		rtPendantUpDownFast(CLK 	:= stCommandsIn.bPendantUpDownFast);
		ftPendantUpDownFast(CLK 	:= stCommandsIn.bPendantUpDownFast);	
		bChangeSpeedUpDown			S= (rtPendantUpDownFast.Q OR ftPendantUpDownFast.Q);
		bChangeSpeedUpDown			R= NOT CartesianZAxisRef.Status.Moving;
	
 CASE 	diManualModeCase OF
	 
		 0:
	mcCatcherHalt.Execute								:=	FALSE;	 
		 
	 	//Ruchy manualne
	mcCartesianYManualMove.JogForward					:= NOT mcCartesianYManualMove.JogBackwards AND NOT bChangeSpeedRightLeft AND
															(bManualCartesianYJogPlus OR stCommandsIn.bPendantRightwardMovement);
	mcCartesianYManualMove.JogBackwards					:= NOT mcCartesianYManualMove.JogForward AND NOT bChangeSpeedRightLeft AND
															(bManualCartesianYJogMinus OR stCommandsIn.bPendantLeftwardMovement);
	mcCartesianYManualMove.Velocity						:= SEL(stCommandsIn.bPendantRightLeftFast, 5.0, 50.0); 
                                            			
	mcCartesianZManualMove.JogForward					:= NOT mcCartesianZManualMove.JogBackwards AND NOT bChangeSpeedUpDown AND
															(bManualCartesianZJogPlus OR stCommandsIn.bPendantUpwardMovement);
	mcCartesianZManualMove.JogBackwards					:= NOT mcCartesianZManualMove.JogForward AND NOT bChangeSpeedUpDown AND
															(bManualCartesianZJogMinus OR stCommandsIn.bPendantDownwardMovement);
	mcCartesianZManualMove.Velocity						:= SEL(stCommandsIn.bPendantUpDownFast, 5.0, 50.0); 
	                                        			
	mcPreScrewerManualMove.JogForward					:= bManualPreScrewerJogPlus;
	mcPreScrewerManualMove.JogBackwards					:= bManualPreScrewerJogMinus;
	mcPreScrewerManualMove.Velocity						:= 90;
                                            			
	mcCatcherManualMove.JogForward						:= bManualCatcherJogPlus;
	mcCatcherManualMove.JogBackwards					:= bManualCatcherJogMinus;
	mcCatcherManualMove.Velocity						:= 15; 
	                                        			
	bCapSucker[1]											:= bManualCapSucker1;	
	bCapSucker[2]											:= bmanualCapSucker2;	
	bCapSucker[3]											:= bManualCapSucker3;	
	bCapSucker[4]											:= bManualCapSucker4;	
	                          	    					                     
	bCapBlower1											:= bManualCapBlower1;	
	bCapBlower2											:= bManualCapBlower2;	
	bCapBlower3											:= bManualCapBlower3;	
	bCapBlower4											:= bManualCapBlower4;	
	                          		    				                 
	bCapCatcher1										:= bManualCapCatcher1;
	bCapCatcher2										:= bManualCapCatcher2;
	bCapCatcher3										:= bManualCapCatcher3;
	bCapCatcher4					    				:= bManualCapCatcher4;
	
	
	
	IF bManualStrawCatchersOpen	THEN
		bStrawCatchersOpen								:= TRUE;
		bStrawCatchersClose								:= FALSE;
		bManualStrawCatchersClose						:= FALSE;
	END_IF	                                    		
                                                		
	IF bManualStrawCatchersClose	THEN        		
		bStrawCatchersOpen								:= FALSE;
		bStrawCatchersClose								:= TRUE;
		bManualStrawCatchersOpen						:= FALSE;
	END_IF		                                		
	                                            		
     IF bManualStrawCatcherActuatorOut THEN     		
		 bStrawCatcherActuatorOut						:= TRUE;
		 bStrawCatcherActuatorIn						:= FALSE;
		 bManualStrawCatcherActuatorIn					:= FALSE;
	 END_IF                                     		
	                                            	
     IF bManualStrawCatcherActuatorIn THEN      	
		 bStrawCatcherActuatorIn						:= TRUE;
		 bStrawCatcherActuatorOut						:= FALSE;
		 bManualStrawCatcherActuatorOut					:= FALSE;
	 END_IF
	 
	 //Zaczynam sekwencje 
	 IF trStepButton.Q THEN
		 VirtualEna											:= TRUE;
		 ResetCommands();
		 bCapCatcher1										:= FALSE;
		 bCapCatcher2										:= false;
		 bCapCatcher3										:= false;
		 bCapCatcher4										:= false;
		 bCartesianReady									:= bCartesianInHomePos;
		 diManualModeCase									:= diManualModeCase + 10;
	 END_IF
	 
	 IF rtSetEncoderOffsetAxisZ.Q THEN
		diManualModeCase									:= diManualModeCase + 500;
	 END_IF
 
 
 		10:	//Dojazd do poz home
	bStepButton												:= TRUE;
	                                                    	
	mcCartesianZMoveAbsolute.Execute						:= NOT bAxisZInHomePos;		
	mcCartesianZMoveAbsolute.Position						:= 420;
	mcCartesianZMoveAbsolute.Acceleration					:= 200.0;
	mcCartesianZMoveAbsolute.Deceleration					:= 200.0;
	mcCartesianZMoveAbsolute.Velocity						:= 30;
	                                        				
	//najpierw os Z potem winda chwytakow   				
	mcCatcherMoveAbsolute.Execute							:= NOT bAxisStrawCatcherHomePos AND bAxisZInHomePos;		
	mcCatcherMoveAbsolute.Position							:= stParameters.lrCatcherCatchingPosition;
	mcCatcherMoveAbsolute.Acceleration						:= 200.0;
	mcCatcherMoveAbsolute.Deceleration						:= 200.0;
	mcCatcherMoveAbsolute.Velocity							:= 30;
	                                        				
	mcCartesianYMoveAbsolute.Execute						:= NOT bAxisYInHomePos AND bAxisZInHomePos;
	mcCartesianYMoveAbsolute.Position						:= stParameters.lrPickYPosition;
	mcCartesianYMoveAbsolute.Acceleration					:= 200.0;
	mcCartesianYMoveAbsolute.Deceleration					:= 200.0;
	mcCartesianYMoveAbsolute.Velocity						:= 30; 
	                                                    	
	IF bAxisZInHomePos THEN
		GVL_VIS.bCapSorterPreScrewerCatchStationHoming			:= NOT fbStrawCatcherLift.bHomingDone;
		GVL_VIS.bCapSorterPreScrewerCatcherStationHeightSet		:= NOT GVL_VIS.bCapSorterPreScrewerCatchStationHoming AND NOT bStrawCatcherLiftInHomePos;
		bEnableLift												:= GVL_VIS.bCapSorterPreScrewerCatcherStationHeightSet;
	END_IF

		IF 	bCartesianInHomePos AND bStrawCatcherLiftInHomePos THEN
			mcCartesianZMoveAbsolute.Execute              	:= FALSE;
			mcCatcherMoveAbsolute.Execute                 	:= FALSE;
			mcCartesianYMoveAbsolute.Execute              	:= FALSE;
			GVL_VIS.bCapSorterPreScrewerCatchStationHoming	:= FALSE;
			diManualModeCase								:= diManualModeCase + 5;
		END_IF
		
		15: //Ustaw obracarkę w pozycji
	bStepButton												:= TRUE;
	                                                    	
	mcPreScrewerMoveRelative.Execute						:= TRUE;
	mcPreScrewerMoveRelative.Distance						:=  -1 * DINT_TO_LREAL(LREAL_TO_DINT(PreScrewerAxisRef.NcToPlc.SetPos) MOD 360);
	mcPreScrewerMoveRelative.Acceleration					:= 200.0;
	mcPreScrewerMoveRelative.Deceleration					:= 200.0;
	mcPreScrewerMoveRelative.Velocity						:= 180.0;	
	                                                    	
		IF mcPreScrewerMoveRelative.Done THEN           	
			mcPreScrewerMoveRelative.Execute				:= FALSE;
			
			IF bCartesianReady THEN
				diManualModeCase							:= diManualModeCase + 10;
			ELSE	                                        
				bStepButton									:= FALSE;
				diManualModeCase							:= diManualModeCase + 5;
			END_IF
			
		END_IF	

		
//--------------------------------jazda na poz pick------------------------------------------------------------------			
		20:	//Kolejny krok
	 IF trStepButton.Q THEN
		diManualModeCase									:= diManualModeCase + 5;
	 END_IF

		25:
	bStepButton												:= TRUE;
	
	mcCartesianZMoveAbsolute.Execute						:= TRUE;		
	mcCartesianZMoveAbsolute.Position						:= stParameters.lrPickZPosition;
	
		IF mcCartesianZMoveAbsolute.Done THEN
			mcCartesianZMoveAbsolute.Execute				:= FALSE;
			bStepButton										:= FALSE;
			diManualModeCase								:= diManualModeCase + 5;
		END_IF

		
//----------------------------Sekwencyjne zalączanie ssawek----------------------------------------------------------------	
		30: //Kolejny krok
	 IF trStepButton.Q THEN
		FOR i:=1 TO 4 DO
			bCapSucker[i]									:= TRUE;
		END_FOR	 
	 
		diManualModeCase									:= diManualModeCase + 5;
	 END_IF
		
		35: //Załączanie ssawek
	tonVacuumWatchdog.IN									:= TRUE;
	bStepButton												:= TRUE;

	
	
		IF tonVacuumWatchdog.Q THEN	
			bStepButton										:= FALSE;		 
			tonVacuumWatchdog.IN							:= FALSE;								
			diManualModeCase								:= diManualModeCase + 20;				
		END_IF
		
		
//-------------------------------Dojazd do pozycji zamykania wings'ów-------------------------------------------------------------------			
		55: //Kolejny krok
	 IF trStepButton.Q THEN
		diManualModeCase									:= diManualModeCase + 5;
	 END_IF	
	 
	 	60:
	bStepButton												:= TRUE;	
	mcCartesianZMoveAbsolute.Execute						:= TRUE;		
	mcCartesianZMoveAbsolute.Position						:= stParameters.lrCapCatcherZPosition;	
		
		IF mcCartesianZMoveAbsolute.Done THEN
			
			FOR i:=1 TO 4 DO
				bCapSucker[i]								R= NOT  bCapSucker[i];
			END_FOR 
			
			bStepButton										:= FALSE;	
			mcCartesianZMoveAbsolute.Execute				:= FALSE;
			diManualModeCase								:= diManualModeCase + 5;		
		END_IF

		
//--------------------------------Zamykanie vings'ów------------------------------------------------------------------			
		65://Kolejny krok
	 IF trStepButton.Q THEN
		diManualModeCase									:= diManualModeCase + 5;
	 END_IF	
	 
	 	70:
	bStepButton												:= FALSE;	
	bCapCatcher1											:= TRUE;
	bCapCatcher2											:= TRUE;
	bCapCatcher3											:= TRUE;
	bCapCatcher4											:= TRUE;
	diManualModeCase										:= diManualModeCase + 5;

	
//---------------------------------dojazd do poz. Top-----------------------------------------------------------------			
		75://Kolejny krok
	 IF trStepButton.Q THEN
		diManualModeCase									:= diManualModeCase + 5;
	 END_IF	
		
		80:
	bStepButton												:= TRUE;
	mcCartesianZMoveAbsolute.Execute						:= TRUE;
	mcCartesianZMoveAbsolute.Position						:= stParameters.lrTopZPosition;
		
		IF mcCartesianZMoveAbsolute.Done THEN
			bStepButton										:= FALSE;	
			mcCartesianZMoveAbsolute.Execute				:= FALSE;
			diManualModeCase								:= diManualModeCase + 5;		
		END_IF

		
//-----------------------------------dojazd osi Y do pozycji place---------------------------------------------------------------			
		85://Kolejny krok
	 IF trStepButton.Q THEN
		diManualModeCase									:= diManualModeCase + 5;
	 END_IF	
	 
	 90:
	bStepButton												:= TRUE;
	mcCartesianYMoveAbsolute.Execute						:= TRUE;
	mcCartesianYMoveAbsolute.Position						:= stParameters.lrPlaceYPosition;
	
	 mcCartesianZMoveAbsolute.Execute						:= CartesianYAxisRef.NcToPlc.ActPos > stParameters.lrPickYPosition + 50.0;
	 mcCartesianZMoveAbsolute.Position						:= stParameters.lrCartesianCatchZPosition;
	 
		IF mcCartesianYMoveAbsolute.Done AND mcCartesianZMoveAbsolute.Done THEN
			bStepButton										:= FALSE;
			mcCartesianYMoveAbsolute.Execute				:= FALSE;
			GVL_VIS.bCapSorterPreScrewerBottleCatcherCatch	:= TRUE;					//Zamykanie chwytaków butelek
			diManualModeCase								:= diManualModeCase + 10;
		END_IF		
		
		
		
		

		
//-------------------------------Wybór pracy: słomka albo fliptop & sterowanie krabami------------------------	
		100://Kolejny krok
	 IF trStepButton.Q THEN
		diManualModeCase									:= diManualModeCase + 5;
	 END_IF	
	 
		105://Ustaw pozycję wirtualnej osi tak samo jak na osi Z
	fbVirtualAxis.fPosition									:= CartesianZAxisRef.NcToPlc.ActPos;
	fbVirtualAxis.SetPosAbsClearLag(bExecute				:= TRUE);
		
		IF fbVirtualAxis.pSetPos.Busy THEN
			diManualModeCase								:= diManualModeCase + 1;
		ELSIF fbVirtualAxis.pSetPos.Error OR fbVirtualAxis.pSetPos.CommandAborted THEN
    		udiErrorID										:= 6;
    		udiErrorID										:= udiErrorID + iStationIndex;
    		sErrorDescription								:= 'Błąd podnosnika lub brak zasilania';
    		sErrorDescription2								:= ' ';	
		END_IF
		
		106:
	fbVirtualAxis.SetPosAbsClearLag(bExecute				:= FALSE);
		
		IF fbVirtualAxis.pSetPos.Done THEN
			diManualModeCase								:= diManualModeCase + 4;
		END_IF


		110: 	//Przy aktywowanych slomkach--> wysuń kraby
	IF stParameters.bStrawCatcherON THEN
		bStrawCatcherActuatorIn								:= FALSE;
		bStrawCatcherActuatorOut							:= TRUE; 
		diManualModeCase									:= diManualModeCase + 1;
	ELSE
			//przeskakuję do sprawdzania czy mam szukanie gwintu
		bStrawCatcherActuatorIn								:= TRUE;
		bStrawCatcherActuatorOut							:= FALSE; 			
		fbGearInAxisZ.Enable								:= TRUE;
		
			IF fbGearInAxisZ.InGear THEN
				fbGearInAxisZ.Enable						:= FALSE;
				IF stParameters.lrScrewFinding > 0 THEN
			 		diManualModeCase						:= diManualModeCase + 26;
		 		ELSE
					diManualModeCase						:= diManualModeCase + 30;
			 	END_IF
			 END_IF
	END_IF
		
		
		111://zamknij kraby
	bStepButton												:= TRUE;	
	bStrawCatchersOpen										:= NOT bStrawCatcherOut;
	bStrawCatchersClose										:= bStrawCatcherOut;
	
		//zamkniete kraby
		IF tonStrawCatcher1Close.Q (*AND tonStrawCatcher2Close.Q*) AND tonStrawCatcher3Close.Q AND tonStrawCatcher4Close.Q THEN
			bStepButton										:= FALSE;
			diManualModeCase								:= diManualModeCase + 4;
		END_IF

		
//-----------------------------------Prowadzenie slomki do pozycji wspolnego ruchu-------------------------------			
		115://Kolejny krok
	 IF trStepButton.Q THEN
		diManualModeCase									:= diManualModeCase + 5;
	 END_IF			
		
		120://gear'owanie napędu prowadzenia słomki
	fbGearInCatcherAxis.Enable								:= TRUE;
	fbGearInCatcherAxis.GearRatio							:= 1;
	fbGearInAxisZ.Enable									:= TRUE;
	fbGearInAxisZ.GearRatio									:= 0.0000000001;
	bStepButton												:= TRUE;
		
		IF fbGearInCatcherAxis.InGear AND fbGearInAxisZ.InGear THEN
			//fbGearInCatcherAxis.Enable						:= FALSE;
			//fbGearInAxisZ.Enable							:= FALSE;
			diManualModeCase								:= diManualModeCase + 10;
		END_IF

		
//-----------------------------------Prowadzenie, wkładanie nasadki oraz rozgirowanie osi do prowadzenia słomki------------------------------------------			
		130: 
	fbVirtualAxis.fPosition									:= (stParameters.LrCheckStrawCatcherActuatorZPosition - stParameters.lrStrawInsertDistance);	//Pozycja sprawdzania cofnięcia krabów
	fbVirtualAxis.fVelocity									:= 100.0;	//10
	fbVirtualAxis.fAcceleration								:= 1000.0;
	fbVirtualAxis.fDeceleration								:= 1000.0;
	fbVirtualAxis.fJerk										:= 10000.0;			
			
	bStepButton												:= TRUE;
	bVirtualMove											:= TRUE;				
//	fbGearInAxisZ.Execute									:= CatcherAxisRef.NcToPlc.ActPos <= (stParameters.lrCatcherPlacePosition + stParameters.lrStrawInsertDistance);

	//IF CatcherAxisRef.NcToPlc.ActPos <= (stParameters.lrCatcherCatchingPosition - stParameters.lrStrawInsertDistance) THEN
	//	fbGearInAxisZ.GearRatio								:= 1;
	//END_IF
	
	IF (CatcherAxisRef.NcToPlc.ActPos + stParameters.lrCatcherHightSV) <= (stParameters.lrCartesianCatchZPosition-(stParameters.lrCapHight + 25)) THEN
		fbGearInAxisZ.GearRatio								:= 1;
	END_IF
	
			//Otwórz chwytaki słomek
		IF CartesianZAxisRef.NcToPlc.ActPos <= stParameters.lrStrawCatcherZPosition THEN					
			bStrawCatchersOpen								:= TRUE;
			bStrawCatchersClose								:= FALSE;
		END_IF
		
		// 10mm stały offset - wysokość nad butelką
		IF (CatcherAxisRef.NcToPlc.ActPos <= 1.0) OR (CatcherAxisRef.NcToPlc.ActPos + 32 <= ((stParameters.lrBottleHight + 10.0) - stParameters.lrCatcherHightSV)) THEN	//13 20
			fbGearInCatcherAxis.GearRatio					:= 0.0000000001;
		END_IF
	
			IF tonStrawCatcher1Open.Q AND tonStrawCatcher2Open.Q AND tonStrawCatcher3Open.Q AND tonStrawCatcher4Open.Q THEN																				
				//Cofnij chwytaki słomek
				bStrawCatcherActuatorIn						:= TRUE;
				bStrawCatcherActuatorOut					:= FALSE;				
			END_IF			
			
				IF stVirtualMove_Out.Done THEN
					//fbGearInAxisZ.Enable					:= FALSE;
					//fbGearOutCatcherAxis.Execute			:= FALSE;
					fbGearInCatcherAxis.GearRatio				:= 0.0000000001;
					bVirtualMove							:= FALSE;	
					bStepButton								:= FALSE;
					diManualModeCase						:= diManualModeCase + 5;
				END_IF					
		
//------------------------------------Zakończenie wkładania nasadki---------------------------------------------------			
		135://Kolejny krok
		//mcCatcherHalt.Execute								:=	FALSE;
		
	 IF trStepButton.Q THEN
		 IF stParameters.lrScrewFinding > 0 THEN
			 diManualModeCase								:= diManualModeCase + 1;
		 ELSE
			 diManualModeCase								:= diManualModeCase + 5;
		 END_IF
		
	 END_IF	

//------------------------------------Szukanie gwintu---------------------------------------------------				 	
		136:
	fbVirtualAxis.fVelocity									:= 800.0;	//10
	fbVirtualAxis.fAcceleration								:= 1000.0;
	fbVirtualAxis.fDeceleration								:= 1000.0;
	fbVirtualAxis.fJerk										:= 10000.0;			
		
	fbVirtualAxis.fPosition									:= stParameters.lrScrewerStartZPosition;
	bVirtualMove											:= TRUE;
	bStepButton												:= TRUE;	
	
		IF stVirtualMove_Out.Done THEN
			bCapSucker[1]										:= FALSE;
			bCapSucker[2]										:= FALSE;
			bCapSucker[3]										:= FALSE;
			bCapSucker[4]										:= FALSE;

			mcPreScrewerMoveRelative.Distance				:= stParameters.lrScrewFinding * -1.0;
			mcPreScrewerMoveRelative.Acceleration			:= stParameters.lrScrewAcceleration;
			mcPreScrewerMoveRelative.Deceleration			:= stParameters.lrScrewAcceleration;
			mcPreScrewerMoveRelative.Velocity				:= stParameters.lrScrewSpeed;
			mcPreScrewerMoveRelative.Execute				:= TRUE;
		END_IF
		
				IF mcPreScrewerMoveRelative.Done OR ABS(PreScrewerAxisRef.NcToPlc.PosDiff) > 60.0 OR mcPreScrewerMoveRelative.Error THEN
					bVirtualMove							:= FALSE;
					bStepButton								:= FALSE;
					mcPreScrewerMoveRelative.Execute		:= FALSE;
					diManualModeCase						:= diManualModeCase + 1;
				END_IF	
		
		137://Kolejny krok
	 IF trStepButton.Q THEN
		 diManualModeCase									:= diManualModeCase + 3;		
	 END_IF					
	 
	 	140:
	lrPreScrewerAxisSavedPosition							:= PreScrewerAxisRef.NcToPlc.ActPos;	//zapisywanie pozycji przed zakrecaniem		
	fbVirtualAxis.fPosition									:= stParameters.lrPlaceZPosition - stParameters.lrStrawInsertDistance;
	fbVirtualAxis.fVelocity									:= stParameters.lrCatcherSpeed;
	fbVirtualAxis.fAcceleration								:= 1000.0;
	fbVirtualAxis.fDeceleration								:= 1000.0;
	fbVirtualAxis.fJerk										:= 10000.0;
	bVirtualMove											:= TRUE;
	bStepButton												:= TRUE;
	
		IF CartesianZAxisRef.NcToPlc.ActPos <= stParameters.lrScrewerStartZPosition + 1.0 THEN
			bCapSucker[1]										:= FALSE;
			bCapSucker[2]										:= FALSE;
			bCapSucker[3]										:= FALSE;
			bCapSucker[4]										:= FALSE;
			mcPreScrewerMoveRelative.Execute				:= TRUE;
			mcPreScrewerMoveRelative.Distance				:= stParameters.lrScrewDistance;
			mcPreScrewerMoveRelative.Acceleration			:= stParameters.lrScrewAcceleration;
			mcPreScrewerMoveRelative.Deceleration			:= stParameters.lrScrewAcceleration;
			mcPreScrewerMoveRelative.Velocity				:= stParameters.lrScrewSpeed;// do bylo 600.0;//stParameters.lrScrewSpeed;
			diManualModeCase								:= diManualModeCase + 5;			
		END_IF

	
		145:
	bStepButton												:= TRUE;
	
			//otwórz centrowniki butelek
		IF (GVL_Recipe.bCapSorterPreScrewerCatchAngleOpenEnaShow AND
			ABS(PreScrewerAxisRef.NcToPlc.ActPos - lrPreScrewerAxisSavedPosition) >= GVL_Recipe.lrCapSorterPreScrewerCatchAngleOpenSV) THEN
			bBottleCatcherCatchTemp					:= FALSE;
		END_IF
	
		IF PreScrewerAxisRef.NcToPlc.PosDiff > 100.0 OR (stVirtualMove_Out.Done AND mcPreScrewerMoveRelative.Done) THEN
			bBottleCatcherCatchTemp							:= FALSE;
			bCapCatcher1									:= FALSE;
		 	bCapCatcher2									:= FALSE;
		 	bCapCatcher3									:= FALSE;
		 	bCapCatcher4									:= FALSE;
			bVirtualMove									:= FALSE;
			bCapsBlowON										:= TRUE;
			
				IF fbVirtualAxis.bMoving THEN
					fbVirtualAxis.Halt(bExecute := TRUE);
				ELSE
					fbVirtualAxis.Halt(bExecute := FALSE);
					diManualModeCase						:= diManualModeCase + 5;
				END_IF	
				
		END_IF
		
		150:
	bStepButton												:= TRUE;	
	fbVirtualAxis.fPosition									:= stParameters.lrPlaceZPosition + 20.0;	
	fbVirtualAxis.fVelocity									:= 800.0;//10.0;
	fbVirtualAxis.fAcceleration								:= 1000.0;
	fbVirtualAxis.fDeceleration								:= 1000.0;
	fbVirtualAxis.fJerk										:= 10000.0;
	bVirtualMove											:= TRUE;
	fbGearInCatcherAxis.Enable								:= FALSE;
	fbGearInAxisZ.Enable									:= FALSE;
	
		IF stVirtualMove_Out.Done THEN
			bVirtualMove									:= FALSE;
			diManualModeCase								:= diManualModeCase + 5;
		END_IF
		
		
					151:		//na testy do usunięcia
					fbVirtualAxis.fPosition									:= CartesianZAxisRef.NcToPlc.ActPos;
					fbVirtualAxis.SetPosAbsClearLag(bExecute				:= TRUE);
					
					152:
					fbVirtualAxis.SetPosAbsClearLag(bExecute				:= FALSE);
	
	
		155:
	fbGearOutAxisZ.Execute									:= TRUE;
	fbGearOutCatcherAxis.Execute							:= TRUE;
	
		IF NOT CartesianZAxisRef.Status.Coupled AND NOT CatcherAxisRef.Status.Coupled THEN
			fbGearOutAxisZ.Execute							:= FALSE;
			fbGearOutCatcherAxis.Execute					:= FALSE;
			bStepButton										:= FALSE;
			diManualModeCase								:= diManualModeCase + 5;
		END_IF

//-------------------------------------Dojazd do poz home---------------------------------------------			
		160://Kolejny krok
	 IF trStepButton.Q THEN
		diManualModeCase									:= diManualModeCase + 5;
	 END_IF	
		
		165:
	GVL_VIS.bCapSorterPreScrewerBottleCatcherCatch	:= FALSE;	
	bStepButton										:= TRUE;	
	mcCartesianZMoveAbsolute.Execute				:= TRUE;		
	mcCartesianZMoveAbsolute.Position				:= stParameters.lrTopZPosition;
                                            		
	mcCartesianYMoveAbsolute.Execute				:= ABS(mcCartesianZMoveAbsolute.Position - stParameters.lrTopZPosition) <= 1.0;
	mcCartesianYMoveAbsolute.Position				:= stParameters.lrPickYPosition;
	                                        		
	mcPreScrewerMoveRelative.Execute				:= mcCartesianYMoveAbsolute.Done;
	mcPreScrewerMoveRelative.Velocity				:= 180.0;
	mcPreScrewerMoveRelative.Distance				:= -1 * DINT_TO_LREAL(LREAL_TO_DINT(PreScrewerAxisRef.NcToPlc.SetPos) MOD 360);
	                                        		
	mcCatcherMoveAbsolute.Execute					:= mcCartesianZMoveAbsolute.Done;		
	mcCatcherMoveAbsolute.Position					:= stParameters.lrCatcherCatchingPosition;
	
		IF (mcCartesianZMoveAbsolute.Done AND mcCartesianYMoveAbsolute.Done
			AND mcPreScrewerMoveRelative.Done AND mcCatcherMoveAbsolute.Done) THEN
				bCapsBlowON							:= TRUE;
				bStepButton							:= FALSE;
				ResetCommands();            		
				diManualModeCase					:= 0;
		END_IF	 
		
		
	500: //Ustawianie offsetu na soi Z kartezjana
	bCartesianZServoPower				:= FALSE;
	
	fbAxisZPositioningOffset.Position	:= 0.0;
	fbAxisZPositioningOffset.Execute	:= NOT CartesianZAxisRef.Status.Disabled;
	
	IF fbAxisZPositioningOffset.Busy THEN
		diManualModeCase				:= diManualModeCase + 5;
	END_IF
		
	505:
	IF NOT fbAxisZPositioningOffset.Busy THEN
		fbAxisZPositioningOffset.Execute := FALSE;
		bCartesianZServoPower			 := TRUE;
		diManualModeCase				:= diManualModeCase + 5;
	END_IF
	
	510:
	IF 	mcCartesianZPower.Status THEN
		diManualModeCase				:= 0;
	END_IF
		
 END_CASE
END_ACTION

ACTION PreparingToDisable:
//BAZOWANIE 

mcCartesianYPower.Override				:=	100;			
mcCartesianZPower.Override				:=	100;			
mcPreScrewerPower.Override				:=	100;			
mcCatcherPower.Override					:=	100;	

bCartesianYServoPower					:= TRUE;
bCartesianZServoPower					:= TRUE;
bPreScrewerPower						:= TRUE;
bCatcherPower							:= TRUE;	

mcCartesianYManualMove.JogBackwards		:=FALSE;
mcCartesianZManualMove.JogBackwards		:=FALSE;
mcPreScrewerManualMove.JogBackwards		:=FALSE;
mcCatcherManualMove.JogBackwards		:=FALSE;

mcCartesianYManualMove.JogForward		:=FALSE;
mcCartesianZManualMove.JogForward		:=FALSE;
mcPreScrewerManualMove.JogForward		:=FALSE;
mcCatcherManualMove.JogForward			:=FALSE;
bCycleNotDone							:= FALSE;



IF mcCartesianYPower.Status AND mcCartesianZPower.Status AND mcPreScrewerPower.Status AND mcCatcherPower.Status THEN
		
		CASE iDisablingCase OF
		
			0:
				iDisablingCase							:= iDisablingCase	+	10;
			
			10: 

				//Otwórz chwytaki
				bCapCatcher1				:= FALSE;
				bCapCatcher2				:= FALSE;
				bCapCatcher3				:= FALSE;
				bCapCatcher4				:= FALSE;
				//Wyłącz ssawki
				bCapSucker[1]				:= FALSE;
				bCapSucker[2]				:= FALSE;
				bCapSucker[3]				:= FALSE;
				bCapSucker[4]				:= FALSE;
				//Wyłącz odmuchy
				bCapBlower1					:= FALSE;
				bCapBlower2					:= FALSE;
				bCapBlower3					:= FALSE;
				bCapBlower4					:= FALSE;
				//Otwórz chwytaki słomek
				bStrawCatchersOpen			:= TRUE;
				bStrawCatchersClose			:= FALSE;
				//Cofnij chwytaki słomek
				bStrawCatcherActuatorIn		:= TRUE;
				bStrawCatcherActuatorOut	:= FALSE;
				//Podjedź robotem i chwytakiem słomek w górę jak cofnięty chwytak słomek - bazuj podnośnik Jisang
				IF tonStrawCatcherIn.Q THEN	
					mcCartesianZMoveAbsolute.Execute		:= TRUE;		
					mcCartesianZMoveAbsolute.Position		:= 420;//stParameters.lrTopZPosition;
					mcCartesianZMoveAbsolute.Acceleration	:= stParameters.lrPickerAcceleration;
					mcCartesianZMoveAbsolute.Deceleration	:= stParameters.lrPickerAcceleration;
					mcCartesianZMoveAbsolute.Velocity		:= 30;//stParameters.lrPickerSpeed;
					
					mcCatcherMoveAbsolute.Execute			:= TRUE;		
					mcCatcherMoveAbsolute.Position			:= stParameters.lrCatcherCatchingPosition;
					mcCatcherMoveAbsolute.Acceleration		:= stParameters.lrCatcherAcceleration;
					mcCatcherMoveAbsolute.Deceleration		:= stParameters.lrCatcherAcceleration;
					mcCatcherMoveAbsolute.Velocity			:= 30;//stParameters.lrCatcherSpeed;

					//Następny krok
					iDisablingCase								:= iDisablingCase + 10;
				END_IF
				//Reset komendy ruchu osi X
				mcCartesianYMoveAbsolute.Execute		:= FALSE;
				
		
			20:		
	(*Czekam na pozycję Z w górze i ruszam osią poziomą X na pozycję pobierania i czekam na obie pozycje*)
				//bStrawCatcherLiftEnable						R= ABS(CartesianYAxisRef.NcToPlc.ActPos - stParameters.lrPickYPosition)<=10.0;
				
				IF (CartesianZAxisRef.NcToPlc.ActPos > stParameters.lrTopZPosition - stParameters.lrBendingDistance) OR
					mcCartesianZMoveAbsolute.Done THEN					
					//Jedź osią poziomą X na pozycję pick
					mcCartesianYMoveAbsolute.Execute		:= TRUE;
					mcCartesianYMoveAbsolute.Position		:= stParameters.lrPickYPosition;
					mcCartesianYMoveAbsolute.Acceleration	:= stParameters.lrPickerAcceleration;
					mcCartesianYMoveAbsolute.Deceleration	:= stParameters.lrPickerAcceleration;
					mcCartesianYMoveAbsolute.Velocity		:= 30;//stParameters.lrPickerSpeed;
					//Ustaw obracarkę w pozycji
					mcPreScrewerMoveRelative.Execute		:= TRUE;
					mcPreScrewerMoveRelative.Distance		:=  -1 * DINT_TO_LREAL(LREAL_TO_DINT(PreScrewerAxisRef.NcToPlc.SetPos) MOD 360);
					mcPreScrewerMoveRelative.Acceleration	:= stParameters.lrScrewAcceleration;
					mcPreScrewerMoveRelative.Deceleration	:= stParameters.lrScrewAcceleration;
					mcPreScrewerMoveRelative.Velocity		:= 180;//stParameters.lrScrewSpeed;
				END_IF
				IF mcPreScrewerMoveRelative.Done THEN
					mcPreScrewerMoveRelative.Execute		:= FALSE;
					mcPreScrewerHome(Axis := PreScrewerAxisRef, HomingMode := MC_Direct, Position := 0, Execute := TRUE);					
				END_IF
				//Jak obie pozycje osiągnięte to następny krok
				IF mcCartesianYMoveAbsolute.Done AND mcCartesianZMoveAbsolute.Done AND mcPreScrewerHome.Done AND fbStrawCatcherLift.eState =  E_Station.eDisabled THEN
					//Reset komendy ruchu osi
					mcCartesianYMoveAbsolute.Execute		:= FALSE;
					mcCartesianZMoveAbsolute.Execute		:= FALSE;
					mcPreScrewerHome.Execute				:= FALSE;
					//Wysuń chwytaki słomek jesli to potrzebuje recepta
					bStrawCatcherActuatorIn					:= TRUE;
					bStrawCatcherActuatorOut				:= FALSE;
					//Następny krok
					iDisablingCase								:= iDisablingCase + 10;
				END_IF
			
			30:	//Koniec
				eState								:= E_Station.eDisabled;
				bHomingDone							:= FALSE;
				iDisablingCase						:= 0;
		END_CASE
END_IF
END_ACTION

ACTION Reject:

CASE iRejectCase OF
	0:

		mcCartesianZMoveAbsolute.Position	:= stParameters.lrPickZPosition - lrAxisZ_RejectOffset;	
		mcCartesianZMoveAbsolute.Execute	:= NOT bTubeReject;
	
				//Przyssanie wszystkich nasadek (przypadek wcisnietej), lub pojedynczej (wykryto brak słomki)
			FOR i:=1 TO 4 DO	
				bCapSucker[i]					:=SEL(bTubeReject, stParameters.bPickerActiv[i] AND NOT tonSuckedOk[i].Q, NOT stMoverStatus.stSlotStatus[i].bTubePresent AND stParameters.bPickerActiv[i]);//SEL(bTubeReject, TRUE, NOT stMoverStatus.stSlotStatus[i].bTubePresent AND stParameters.bPickerActiv[i]);
			END_FOR
		
		iRejectCase	:= 5;
	
	
	5:
			IF bTubeReject OR mcCartesianZMoveAbsolute.Done THEN
				mcCartesianZMoveAbsolute.Execute	:= FALSE;
				iRejectCase	:= 10;
			END_IF
	
	10:
		tonVacuumWatchdog.IN					:= TRUE;
	

		
			IF bAllSlotsVacuumStatus OR tonVacuumWatchdog.Q THEN
					//Podjazd do góry
				mcCartesianZMoveAbsolute.Position	:= stParameters.lrTopZPosition;
				mcCartesianZMoveAbsolute.Execute	:= TRUE;	
				tonVacuumWatchdog.IN				:= FALSE;
				iRejectCase	:= 20;
			END_IF
	
	20:
			//Zamykanie łapek
			IF CartesianZAxisRef.NcToPlc.ActPos > stParameters.lrCapCatcherZPosition THEN
				bCapCatcher1					:= TRUE;
				bCapCatcher2					:= TRUE;
				bCapCatcher3					:= TRUE;
				bCapCatcher4					:= TRUE;
			ELSIF rtAxisZMoving.Q THEN	//oddmuch nie przyssanych nakrętek
				bCapBlow1						:= NOT bCapSucker[1];
            	bCapBlow2						:= NOT bCapSucker[2];
            	bCapBlow3						:= NOT bCapSucker[3];
            	bCapBlow4						:= NOT bCapSucker[4];
				bCapsBlowON						:= TRUE;
			END_IF
			
			IF ABS(CartesianZAxisRef.NcToPlc.ActPos - mcCartesianZMoveAbsolute.Position) <= stParameters.lrBendingDistance THEN
				mcCartesianZMoveAbsolute.Execute	:= FALSE;	
				bMissingCaps						:= TRUE;
				mcCartesianYMoveAbsolute.Position	:= 3.0;
				mcCartesianYMoveAbsolute.Execute	:= TRUE;
				
					FOR i:= 1 TO 4 DO
						bCapSucker[i]				:= FALSE;
					END_FOR				
				
				iRejectCase							:= 30;
			END_IF
		
		30:
			IF ABS(CartesianYAxisRef.NcToPlc.ActPos - mcCartesianYMoveAbsolute.Position) <= stParameters.lrBendingDistance THEN
				mcCartesianYMoveAbsolute.Execute	:= FALSE;
					IF NOT mcCartesianZMoveAbsolute.Busy THEN
						mcCartesianZMoveAbsolute.Position	:= 380.0;
						mcCartesianZMoveAbsolute.Execute	:= TRUE;	
						iRejectCase		:= 40;
					END_IF
			ELSIF ABS(CartesianYAxisRef.NcToPlc.ActPos - mcCartesianYMoveAbsolute.Position) <= 50.0 THEN	
					bCapCatcher1					:=FALSE;
					bCapCatcher2					:=FALSE;
					bCapCatcher3					:=FALSE;
					bCapCatcher4					:=FALSE;
			END_IF
			
		40:
			IF ABS(CartesianZAxisRef.NcToPlc.ActPos - mcCartesianZMoveAbsolute.Position) <= stParameters.lrBendingDistance AND NOT bCapsBlowON THEN
				bCapsBlowON						:= TRUE;
				bCapBlow1						:= TRUE;
            	bCapBlow2						:= TRUE;
            	bCapBlow3						:= TRUE;
            	bCapBlow4						:= TRUE;
				mcCartesianZMoveAbsolute.Execute	:= FALSE;	
				iRejectCase		:= 50;
			END_IF
	
		50:
			mcCartesianZMoveAbsolute2.Position		:= stParameters.lrTopZPosition;
			mcCartesianZMoveAbsolute2.Acceleration	:= stParameters.lrPickerAcceleration;
			mcCartesianZMoveAbsolute2.Deceleration	:= stParameters.lrPickerAcceleration;
			mcCartesianZMoveAbsolute2.Velocity		:= stParameters.lrPickerSpeed;
			mcCartesianZMoveAbsolute2.Execute		:= TRUE;
				
			mcCartesianYMoveAbsolute.Position	:= stParameters.lrPickYPosition;
			mcCartesianYMoveAbsolute.Execute	:= ABS(CartesianZAxisRef.NcToPlc.ActPos - mcCartesianZMoveAbsolute2.Position) <= stParameters.lrBendingDistance;
			
				IF mcCartesianYMoveAbsolute.Busy THEN
					mcCartesianZMoveAbsolute2.Execute		:= FALSE;
					iRejectCase		:= 60;
				END_IF
				
		60:
			IF 	mcCartesianYMoveAbsolute.Done THEN
				mcCartesianYMoveAbsolute.Execute	:= FALSE;
				bRejectDone							:= TRUE;
			END_IF
	
END_CASE
END_ACTION

ACTION ResetCommands:
	iAbortingCASE									:=0;
	iStoppingCase 									:=0;
	iHomingCase										:=0;
	iErrorResseting2								:=0;
	iTestResetting									:=0;
	iCountAborting									:=0;
	iSimulationCase									:=0;
	diManualModeCase								:=0;

	bEnableLift										:= FALSE;
	mcCartesianYManualMove.JogBackwards				:= FALSE;
	mcCartesianZManualMove.JogBackwards				:= FALSE;
	mcPreScrewerManualMove.JogBackwards				:= FALSE;
	mcCatcherManualMove.JogBackwards				:= FALSE;
	bReject											:= FALSE;
	bRejectDone										:= FALSE;
	bTubeReject										:= FALSE;
	                                        		   
	mcCartesianYManualMove.JogForward				:= FALSE;
	mcCartesianZManualMove.JogForward				:= FALSE;
	mcPreScrewerManualMove.JogForward				:= FALSE;
	mcCatcherManualMove.JogForward					:= FALSE;
	                                        		   
	mcCartesianYStop.Execute						:= FALSE;
	mcCartesianZStop.Execute						:= FALSE;
	mcPreScrewerStop.Execute						:= FALSE;
	mcCatcherStop.Execute							:= FALSE;
	                                        		
	                                        		
	mcCartesianYMoveAbsolute.Execute				:= FALSE;
	mcCartesianZMoveAbsolute.Execute				:= FALSE;
	mcCartesianZMoveAbsolute2.Execute				:= FALSE;
	mcPreScrewerMoveAbsolute.Execute				:= FALSE;
//	mcPreScrewerMoveRelative.Execute				:= FALSE;
	mcCatcherMoveAbsolute.Execute					:= FALSE;
	
	
	fbCartesianYHardReset.Execute					:= FALSE;
	fbCartesianZHardReset.Execute					:= FALSE;
	fbPreScrewerHardReset.Execute					:= FALSE;
	fbCatcherHardReset.Execute						:= FALSE;
	mcCartesianYSoftReset.Execute					:= FALSE;
	mcCartesianZSoftReset.Execute					:= FALSE;
	mcPreScrewerSoftReset.Execute					:= FALSE;
	mcPreScrewerStop.Execute						:= FALSE;
	mcCatcherSoftReset.Execute						:= FALSE;
	mcPreScrewerMoveRelative.Execute				:= FALSE;
	                                        		
	tonVacuumWatchdog.IN							:= FALSE;
//	bMissingCaps									:= FALSE;	
	                                        		
	//bManualCapSucker1								:= FALSE;
	//bManualCapSucker2								:= FALSE;
	//bManualCapSucker3								:= FALSE;
	//bManualCapSucker4								:= FALSE;
	                      	    		    		
	bManualCapBlower1								:= FALSE;
	bManualCapBlower2								:= FALSE;
	bManualCapBlower3								:= FALSE;
	bManualCapBlower4								:= FALSE;
	                       		    	    		
	//bManualCapCatcher1								:= FALSE;
	//bManualCapCatcher2								:= FALSE;
	//bManualCapCatcher3								:= FALSE;
	//bManualCapCatcher4					    		:= FALSE;
	                                        		
	bManualStrawCatchersOpen						:= FALSE;
	bManualStrawCatchersClose						:= FALSE;
	                 			            		
	bManualStrawCatcherActuatorOut					:= FALSE;
	bManualStrawCatcherActuatorIn					:= FALSE; 
	GVL_VIS.bCapSorterPreScrewerBottleCatcherCatch	:= FALSE;
	bAdditionalBlow									:= FALSE;
	bBottleCatcherCatchTemp							:= FALSE;
	
	tonWaitInPlacePos.IN							:= FALSE;
	fbGearInAxisZ.Enable							:= FALSE;
	fbGearInCatcherAxis.Enable						:= FALSE;
	bVirtualMove									:= FALSE;

//	mcCatcherHalt.Execute							:= FALSE;	
//	fbCamTableSelectAxisZ.Execute					:= FALSE;
//	fbCamInAxisZ.Execute							:= FALSE;
//	fbCamTableSelectCatcher.Execute					:= FALSE;
//	fbCamInAxisCatcher.Execute						:= FALSE;
//	fbCamOutAxisCatcher.Execute						:= FALSE;
//	fbCamOutAxisZ.Execute							:= FALSE;
	
(*
iCloseGripperBeforeScrewingCASE		:= 0;
iScrewingCase						:= 0;
iScrewing2Case						:= 0;
iStoppingCase 						:= 0;
iPreparingToReadyCase				:= 0;
iHomingCase							:= 0;
iMStep								:= 0;

iErrorResseting2					:= 0;
iErrorResseting3					:= 0;

mcHeight1GearInMultiMaster.Enable	:=	FALSE;
mcHeight1GearOut.Execute			:=	FALSE;
mcHeight1MoveAbsolute.Execute		:=	FALSE;
mcHeight1MoveAbsolute2.Execute		:=	FALSE;
mcHeight1Stop.Execute				:=	FALSE;
mcHeight1ManualMove.JogBackwards	:=	FALSE;
mcHeight1ManualMove.JogForward		:=	FALSE;
mcHeight1SoftReset					(Execute:=FALSE,Axis:=Height1AxisRef);
fbHeight1HardReset					(Execute:=FALSE,Axis:=Height1AxisRef);

mcHeight2GearInMultiMaster.Enable	:=	FALSE;
mcHeight2GearOut.Execute			:=	FALSE;
mcHeight2MoveAbsolute.Execute		:=	FALSE;
mcHeight2MoveAbsolute2.Execute		:=	FALSE;
mcHeight2Stop.Execute				:=	FALSE;
mcHeight2ManualMove.JogBackwards	:=	FALSE;
mcHeight2ManualMove.JogForward		:=	FALSE;
mcHeight2SoftReset					(Execute:=FALSE,Axis:=Height2AxisRef);
fbHeight2HardReset					(Execute:=FALSE,Axis:=Height2AxisRef);

mcWidthMoveAbsolute.Execute			:=	FALSE;
mcWidthStop.Execute					:=	FALSE;
mcWidthManualMove.JogBackwards		:=	FALSE;
mcWidthManualMove.JogForward		:=	FALSE;
mcWidthSoftReset					(Execute:=FALSE,Axis:=Height2AxisRef);
fbWidthHardReset					(Execute:=FALSE,Axis:=Height2AxisRef);

mcMoveAbsolute.Execute				:=	FALSE;			
mcScrewer1MoveAbsolute.Execute		:=	FALSE;
mcScrewer2MoveAbsolute.Execute		:=	FALSE;
mcScrewer1Stop.Execute				:=	FALSE;
mcScrewer2Stop.Execute				:=	FALSE;
mcScrewer1ManualMove.JogBackwards	:=	FALSE;
mcScrewer1ManualMove.JogForward		:=	FALSE;
mcScrewer2ManualMove.JogBackwards	:=	FALSE;
mcScrewer2ManualMove.JogForward		:=	FALSE;
mcScrewer1MoveVelocity.Execute		:=	FALSE;
mcScrewer2MoveVelocity.Execute		:=	FALSE;
mcScrewer1MoveVelocity2.Execute		:=	FALSE;
mcScrewer2MoveVelocity2.Execute		:=	FALSE;
mcScrewer1TorqueControl.Execute		:=	FALSE;
mcScrewer2TorqueControl.Execute		:=	FALSE;


bStepModeMoving						:=	FALSE;
mcScrewer1SoftReset					(Execute:=FALSE,Axis:=Screwing1AxisRef);	
mcScrewer2SoftReset					(Execute:=FALSE,Axis:=Screwing2AxisRef);	
fbScrewer1HardReset					(Execute:=FALSE,Axis:=Screwing1AxisRef);	
fbScrewer2HardReset					(Execute:=FALSE,Axis:=Screwing2AxisRef);	


//bWasPreparePick1					:=	FALSE;
//bWasPreparePick2					:=	FALSE;	
*)
END_ACTION

ACTION Running:

tonVacuumWatchdog(PT	:= stParameters.tTimeVacuumWatchdog);
bStopAllowed	:= eRunningState = E_CapPreScrewer.eReady OR eRunningState = E_CapPreScrewer.eVerticalDownToCatchPos;

//Otwieranie chwytaków
//bBottleCatcherCatchTemp		R= CartesianZAxisRef.NcToPlc.ActPos < stParameters.lrGripperOpenPosition;
GVL_VIS.bCapSorterPreScrewerBottleCatcherCatch	:= bBottleCatcherCatchTemp AND bCapSorterPreScrewerBottleCatcherEnableShow;
	
tonWaitInPlacePos(PT	:= stParameters.tWaitInPlacePos);
//tonWaitInPlacePos(PT 	:= T#200MS);
eLastRunningState	:= eRunningState;

CASE eRunningState OF

//====================================
	
	(*Oczekiwanie na wykonanie pojedynczego cyklu*)
	E_CapPreScrewer.eReady:

		
		IF NOT bCycleDone AND NOT bCycleNotDone THEN  
                                      	
			IF bRun THEN 
				fbVirtualAxis.fAcceleration				:= stParameters.lrPickerAcceleration;	//100_000_000.0;
				fbVirtualAxis.fDeceleration				:= stParameters.lrPickerAcceleration;	//100_000_000.0;
				fbVirtualAxis.fJerk						:= stParameters.lrPickerJerk;// 	1_000_000;//100_000_000_000;  

				iRejectCase					:= 0;
				bRejectDone					:= FALSE;
				bReject						:= FALSE;
				bTubeReject					:= FALSE;
				
				//Przygotuj do cyklu - otwórz chwytaki
				bCapCatcher1				:= FALSE;
				bCapCatcher2				:= FALSE;
				bCapCatcher3				:= FALSE;
				bCapCatcher4				:= FALSE;
	
				//Wyłącz ssawki
				bCapSucker[1]				:= FALSE;
				bCapSucker[2]				:= FALSE;
				bCapSucker[3]				:= FALSE;
				bCapSucker[4]				:= FALSE;
				//Wyłącz odmuchy
				bCapBlower1					:= FALSE;
				bCapBlower2					:= FALSE;
				bCapBlower3					:= FALSE;
				bCapBlower4					:= FALSE;
				bCapsBlowON					:= FALSE;
				//Otwórz chwytaki słomek
				bStrawCatchersOpen			:= TRUE;
				bStrawCatchersClose			:= FALSE;
				//Cofnij chwytaki słomek
				bStrawCatcherActuatorIn		:= TRUE;
				bStrawCatcherActuatorOut	:= FALSE;
				//Podjedź robotem i chwytakiem słomek w górę jak cofnięty chwytak słomek
				IF tonStrawCatcherIn.Q THEN	
										
					mcCartesianZMoveAbsolute.Execute		:= TRUE;		
					mcCartesianZMoveAbsolute.Position		:= stParameters.lrTopZPosition;
					mcCartesianZMoveAbsolute.Acceleration	:= stParameters.lrPickerAcceleration;
					mcCartesianZMoveAbsolute.Deceleration	:= stParameters.lrPickerAcceleration;
					mcCartesianZMoveAbsolute.Velocity		:= stParameters.lrPickerSpeed;
					
					mcCatcherMoveAbsolute.Execute			:= TRUE;		
					mcCatcherMoveAbsolute.Position			:= stParameters.lrCatcherCatchingPosition;
					mcCatcherMoveAbsolute.Acceleration		:= stParameters.lrCatcherAcceleration;
					mcCatcherMoveAbsolute.Deceleration		:= stParameters.lrCatcherAcceleration;
					mcCatcherMoveAbsolute.Velocity			:= stParameters.lrCatcherSpeed;
					
					//Następny krok
					eRunningState						:= E_CapPreScrewer.ePreparingToPick;
					bCycleNotDone						:= TRUE;
					
				END_IF
				//Reset komendy ruchu osi X
				mcCartesianYMoveAbsolute.Execute		:= FALSE;
				
			END_IF
		END_IF
			
	(*Czekam na pozycję Z w górze i ruszam osią poziomą X na pozycję pobierania i czekam na obie pozycje*)
	E_CapPreScrewer.ePreparingToPick:
		IF (CartesianZAxisRef.NcToPlc.ActPos > stParameters.lrTopZPosition - stParameters.lrBendingDistance) OR
			mcCartesianZMoveAbsolute.Done THEN
			//Jedź osią poziomą X na pozycję pick
			mcCartesianYMoveAbsolute.Execute		:= TRUE;
			mcCartesianYMoveAbsolute.Position		:= stParameters.lrPickYPosition;
			mcCartesianYMoveAbsolute.Acceleration	:= stParameters.lrPickerAcceleration;
			mcCartesianYMoveAbsolute.Deceleration	:= stParameters.lrPickerAcceleration;
			mcCartesianYMoveAbsolute.Velocity		:= stParameters.lrPickerSpeed;
			//Nakrętka pobrana z wózka nr.1
			bMover1InPickPos						:= SEL((stParameters.lrPickYPosition-GVL_Recipe.lrCapSorterPreScrewerPickXMover1PositionShow) <= 0.5, FALSE, TRUE);
			
			//Ustaw obracarkę w pozycji
			mcPreScrewerMoveRelative.Distance		:=  -1 * DINT_TO_LREAL((LREAL_TO_DINT(PreScrewerAxisRef.NcToPlc.SetPos)+diPreSCrewerHomePos) MOD 360);
			mcPreScrewerMoveRelative.Execute		:= mcPreScrewerMoveRelative.Distance<>0;
			mcPreScrewerMoveRelative.Acceleration	:= stParameters.lrScrewAcceleration;
			mcPreScrewerMoveRelative.Deceleration	:= stParameters.lrScrewAcceleration;
			mcPreScrewerMoveRelative.Velocity		:= stParameters.lrScrewSpeed;
		END_IF
		//Jak obie pozycje osiągnięte to wysuń chwytak słomek i następny krok
		IF mcCartesianYMoveAbsolute.Done AND mcCartesianZMoveAbsolute.Done AND mcCatcherMoveAbsolute.Done THEN
			IF mcPreScrewerMoveRelative.Done OR mcPreScrewerMoveRelative.Distance =0 THEN
				//Reset komendy ruchu osi
				mcCartesianYMoveAbsolute.Execute		:= FALSE;
				mcCartesianZMoveAbsolute.Execute		:= FALSE;
				mcPreScrewerMoveRelative.Execute		:= FALSE;
				mcCatcherMoveAbsolute.Execute			:= FALSE;
				//Wysuń chwytaki słomek jesli to potrzebuje recepta        
				bStrawCatcherActuatorIn					:= NOT stParameters.bStrawCatcherON;
				bStrawCatcherActuatorOut				:= stParameters.bStrawCatcherON;    
				//Następny krok
				eRunningState							:= E_CapPreScrewer.ePicking;
			END_IF
		END_IF
		
	
	(*Zjeżdzam na osią pionową Z na pozycję chwytania i załączam ssawki*)		
	E_CapPreScrewer.ePicking:
		//Podjedź robotem w górę	
		mcCartesianZMoveAbsolute.Execute			:= TRUE;		
		mcCartesianZMoveAbsolute.Position			:= stParameters.lrPickZPosition;
		mcCartesianZMoveAbsolute.Acceleration		:= stParameters.lrPickerAcceleration;
		mcCartesianZMoveAbsolute.Deceleration		:= stParameters.lrPickerAcceleration;
		mcCartesianZMoveAbsolute.Velocity			:= stParameters.lrPickerSpeed;
		//Czekam na wykonanie ruchu
		IF mcCartesianZMoveAbsolute.Done THEN
			//Reset komendy ruchu osi
			mcCartesianZMoveAbsolute.Execute		:= FALSE;
			
			//Zeruje rejestry oraz załączanie ssawek
			 FOR i:=1 TO 4 DO
				 bCapSucker[i]						:= stParameters.bPickerActiv[i]; 
				 aCapPresence[i] 					:= FALSE;
			 END_FOR
	
			//Następny krok
			eRunningState							:= E_CapPreScrewer.eVacumCheckPart1;
		END_IF
	
	(*Sprawdzam czy zassane i jazda w górę*)	
	E_CapPreScrewer.eVacumCheckPart1:
		
		tonVacuumWatchdog.IN						:= TRUE;
		
		IF tonSuckedOk[1].Q = stParameters.bPickerActiv[1] AND tonSuckedOk[2].Q = stParameters.bPickerActiv[2]
			AND tonSuckedOk[3].Q = stParameters.bPickerActiv[3] AND tonSuckedOk[4].Q = stParameters.bPickerActiv[4] THEN
			tonVacuumWatchdog.IN					:= FALSE;
		
				FOR i:=1 TO 4 DO
					IF stParameters.bPickerActiv[i] AND stParameters.bStrawCatcherON AND NOT stMoverStatus.stSlotStatus[i].bTubePresent THEN
						bReject								:= TRUE;
						bTubeReject							:= TRUE;
						lrAxisZ_RejectOffset				:= 0.0;
					END_IF

					IF bMover1InPlacePos THEN
						diMover1VacuumRetry[i]		:= 0;
					ELSE
						diMover2VacuumRetry[i]		:= 0;
					END_IF	
				END_FOR 
				
			eRunningState 							:= E_CapPreScrewer.eVacumCheckPart2;
	
		ELSIF tonVacuumWatchdog.Q THEN
		
			FOR i:=1 TO 4 DO
				bCapSucker[i]							:= tonSuckedOk[i].Q;
				
				//robimy odrzut jeżeli zostanie wykryto brak słomki
				IF stParameters.bPickerActiv[i] AND stParameters.bStrawCatcherON AND NOT stMoverStatus.stSlotStatus[i].bTubePresent THEN
					bReject								:= TRUE;
					bTubeReject							:= TRUE;
					lrAxisZ_RejectOffset				:= 0.0;
				END_IF
				
						//Detekcja niepobranej nasadki --> odrzut aktywowany opcjonalnie z receptury
					IF stParameters.bPickerActiv[i] AND NOT tonSuckedOk[i].Q AND NOT stParameters.bVacuumDeactivate THEN
						bReject							:= SEL(stParameters.bRejectON, bReject, TRUE);
						lrAxisZ_RejectOffset			:= SEL(stParameters.bRejectON, lrAxisZ_RejectOffset, 13.0);	//offset dodatkowego zjazdu kartezjanem 
						
						IF bMover1InPlacePos THEN
							diMover1VacuumRetry[i]		:= diMover1VacuumRetry[i] + 1;
						ELSE	
							diMover2VacuumRetry[i]		:= diMover2VacuumRetry[i] + 1;
						END_IF
					ELSIF tonSuckedOk[i].Q OR stParameters.bVacuumDeactivate THEN
						IF 	bMover1InPlacePos THEN
							diMover1VacuumRetry[i]		:= 0;
						ELSE
							diMover2VacuumRetry[i]		:= 0;
						END_IF	
					END_IF	
	    	
			END_FOR
				tonVacuumWatchdog.IN					:= FALSE;
				eRunningState 							:= E_CapPreScrewer.eVacumCheckPart2;
	
		END_IF
		
		
	E_CapPreScrewer.eVacumCheckPart2:	
			
		//Jezeli nie jest przyssana zadna nasadka to pdjezdzamy na poz. ready oraz wystawiamy flage bMissingCaps
		IF bReject THEN
			Reject();
				IF bRejectDone THEN				
					eRunningState						:= E_CapPreScrewer.eReady;	
				END_IF		
		ELSIF NOT tonSuckedOk[1].Q AND NOT tonSuckedOk[2].Q AND NOT tonSuckedOk[3].Q AND NOT tonSuckedOk[4].Q THEN
			bCapSucker[1]							:= FALSE;
			bCapSucker[2]							:= False;
			bCapSucker[3]							:= False;
		    bCapSucker[4]							:= False;	
			mcCartesianZMoveAbsolute.Execute		:= TRUE;		
			mcCartesianZMoveAbsolute.Position		:= stParameters.lrTopZPosition;
			mcCartesianZMoveAbsolute.Acceleration	:= stParameters.lrPickerAcceleration;
			mcCartesianZMoveAbsolute.Deceleration	:= stParameters.lrPickerAcceleration;
			mcCartesianZMoveAbsolute.Velocity		:= stParameters.lrPickerSpeed;
			
			IF mcCartesianZMoveAbsolute.Done THEN
				bMissingCaps						:= TRUE;
				bCycleDone;
				mcCartesianZMoveAbsolute.Execute	:= FALSE;
				eRunningState						:= E_CapPreScrewer.eReady;	
			END_IF
			
		ELSE
			mcCartesianZMoveAbsolute.Execute		:= NOT stParameters.bVacuumDeactivate;		
			mcCartesianZMoveAbsolute.Position		:= stParameters.lrTopZPosition;
			mcCartesianZMoveAbsolute.Acceleration	:= SEL(GVL_Recipe.iCapSorterProductType = 0 ,stParameters.lrPickerAcceleration , 150.0);//stParameters.lrPickerAcceleration;
//			mcCartesianZMoveAbsolute.Acceleration	:= stParameters.lrPickerAcceleration;
			mcCartesianZMoveAbsolute.Deceleration	:= stParameters.lrPickerAcceleration;
			mcCartesianZMoveAbsolute.Velocity		:= stParameters.lrPickerSpeed;
			tonCapCatcher.IN						:= FALSE;
			
			IF mcCartesianZMoveAbsolute.Busy OR stParameters.bVacuumDeactivate THEN
				mcCartesianZMoveAbsolute.Execute		:= FALSE;
				eRunningState 							:= E_CapPreScrewer.eTransferingVertical; 
			END_IF
			
        
		END_IF		
			
			//przepisuje do rejestrów nakretki które kartezjan pobrał
			aCapPresence[1] := bCapSucker[1];
			aCapPresence[2] := bCapSucker[2];
			aCapPresence[3] := bCapSucker[3];
			aCapPresence[4] := bCapSucker[4];						

		
		
	(*Jazda w górę, zamknięcie łapek i załączenie jazdy w bok*)	
	E_CapPreScrewer.eTransferingVertical:
		
		IF NOT bCapSucker[1] OR NOT bCapSucker[2] OR NOT bCapSucker[3] OR NOT bCapSucker[4] THEN
            bCapBlow1						:= NOT bCapSucker[1];
            bCapBlow2						:= NOT bCapSucker[2];
            bCapBlow3						:= NOT bCapSucker[3];
            bCapBlow4						:= NOT bCapSucker[4];						
			bCapsBlowON						:= TRUE;
		END_IF
		
		//Kleją się kulki 
		IF NOT stParameters.bVacuumDeactivate THEN					
			IF CartesianZAxisRef.NcToPlc.ActPos > stParameters.lrPickZPosition + 10.0 THEN
				mcCartesianZMoveAbsolute2.Execute		:= NOT stParameters.bVacuumDeactivate;		
				mcCartesianZMoveAbsolute2.Position		:= stParameters.lrTopZPosition;
				mcCartesianZMoveAbsolute2.Acceleration	:= stParameters.lrPickerAcceleration;
				mcCartesianZMoveAbsolute2.Deceleration	:= stParameters.lrPickerAcceleration;
				mcCartesianZMoveAbsolute2.Velocity		:= stParameters.lrPickerSpeed;
			END_IF
		END_IF


		IF CartesianZAxisRef.NcToPlc.ActPos > stParameters.lrCapCatcherZPosition OR (CartesianZAxisRef.NcToPlc.ActPos > stParameters.lrTopZPosition - stParameters.lrBendingDistance) THEN
			bCapCatcher1							:= TRUE;
			bCapCatcher2							:= true;
			bCapCatcher3							:= true;
			bCapCatcher4							:= true;
			tonCapCatcher.IN						:= stParameters.bVacuumDeactivate;
		END_IF	
		
		mcCartesianZMoveAbsolute.Execute		:= tonCapCatcher.Q;	
		
		//Dodać sprawdzenie czy gotowy chwytak słomek !!!!!
		//Sprawdzenie pozycji osi pionowej Z i czy wysunięty siłownik chwytaka słomek
		IF ((CartesianZAxisRef.NcToPlc.ActPos > stParameters.lrTopZPosition - stParameters.lrBendingDistance) OR
			mcCartesianZMoveAbsolute.Done) AND (tonStrawCatcherOut.Q OR NOT stParameters.bStrawCatcherON) THEN
			//Jedź osią poziomą X na pozycję pick
				mcCartesianZMoveAbsolute2.Execute		:= FALSE;
				bCapsBlowON								:= FALSE;
				eRunningState 							:= E_CapPreScrewer.eTransferingHorizontal;
				tonCapCatcher.IN						:= FALSE;
		END_IF
	
	(*Przejazd w poziomie*)	
	E_CapPreScrewer.eTransferingHorizontal:	
	
			bCapCatcher1							:= TRUE;//bCapSucker1;
			bCapCatcher2							:= TRUE;//bCapSucker2;
			bCapCatcher3							:= TRUE;//bCapSucker3;
			bCapCatcher4							:= TRUE;//bCapSucker4;
	
		mcCartesianYMoveAbsolute.Position			:= stParameters.lrPlaceYPosition;
		mcCartesianYMoveAbsolute.Acceleration		:= stParameters.lrPickerAcceleration;
		mcCartesianYMoveAbsolute.Deceleration		:= stParameters.lrPickerAcceleration;
		mcCartesianYMoveAbsolute.Velocity			:= stParameters.lrPickerSpeed;
		mcCartesianYMoveAbsolute.Execute			:= TRUE;
		
		IF (CartesianYAxisRef.NcToPlc.ActPos > 200.0 (*stParameters.lrPlaceYPosition - stParameters.lrBendingDistance*)) OR
			mcCartesianYMoveAbsolute.Done AND NOT mcCartesianZMoveAbsolute.Execute THEN			

			//Podjedź robotem w dól	
			mcCartesianZMoveAbsolute.Execute			:= TRUE;		
			mcCartesianZMoveAbsolute.Position			:= stParameters.lrCartesianCatchZPosition;
			mcCartesianZMoveAbsolute.Acceleration		:= stParameters.lrPickerAcceleration;
			mcCartesianZMoveAbsolute.Deceleration		:= stParameters.lrPickerAcceleration;
			mcCartesianZMoveAbsolute.Velocity			:= stParameters.lrPickerSpeed;
		END_IF
		
		//Jak obie pozycje osiągnięte 
		IF mcCartesianZMoveAbsolute.Done THEN
			mcCartesianZMoveAbsolute.Execute		:= FALSE;
		END_IF
			
		//Jak ak obie pozycje osiągnięte to zamykamy chwytaki i następny krok
		IF stParameters.bStrawCatcherON AND CartesianYAxisRef.NcToPlc.ActPos >= stParameters.lrPlaceYPosition THEN
			//Zamknij chwytaki słomek
			bStrawCatchersOpen						:= FALSE;
			bStrawCatchersClose						:= TRUE;	
		END_IF
		
			
		IF  mcCartesianYMoveAbsolute.Done AND mcCartesianZMoveAbsolute.Done THEN
			//Reset komendy ruchu osi
			mcCartesianYMoveAbsolute.Execute		:= FALSE;
			mcCartesianZMoveAbsolute.Execute		:= FALSE;
			
				//Ustaw pozycję wirtualnej osi tak samo jak na osi Z
			fbVirtualAxis.fPosition						:= CartesianZAxisRef.NcToPlc.ActPos;
			fbVirtualAxis.SetPosAbsClearLag(bExecute	:= TRUE);
				
				IF fbVirtualAxis.pSetPos.Busy THEN
					//Następny krok
					eRunningState						:= E_CapPreScrewer.eVerticalDownToCatchPos;	
				END_IF
		END_IF		
		
	(*Przejazd w dól do pozycji chwytanija rurki*)		
	E_CapPreScrewer.eVerticalDownToCatchPos:
		fbVirtualAxis.SetPosAbsClearLag(bExecute				:= FALSE);
		
		//Jak ak obie pozycje osiągnięte to zamykamy chwytaki i następny krok
		IF stParameters.bStrawCatcherON THEN
			//Zamknij chwytaki słomek
			bStrawCatchersOpen						:= FALSE;
			bStrawCatchersClose						:= TRUE;	
		END_IF
				
		IF tonPlacePermission.Q AND ((bCapCatcher1 OR NOT bCapCatcher1) AND (bCapCatcher2  OR NOT bCapCatcher2) AND
									(bCapCatcher3  OR NOT bCapCatcher3) AND(bCapCatcher4  OR NOT bCapCatcher4)) AND (tonStrawCatcher1Close.Q OR NOT stParameters.bStrawCatcherON) THEN				
				bCapCatcher1						:= TRUE;
				bCapCatcher2						:= TRUE;
				bCapCatcher3						:= TRUE;
				bCapCatcher4						:= TRUE;						
				eRunningState						:= E_CapPreScrewer.eAxisGearIn;
		END_IF
		
			//Następny krok
			//IF stParameters.bStrawCatcherON THEN
			//	eRunningState						:= E_CapPreScrewer.eCatching;	
			//ELSE
			//	eRunningState						:= E_CapPreScrewer.ePlacing;	
			//END_IF				
		//END_IF
	
	
	E_CapPreScrewer.eAxisGearIn:
		fbGearInCatcherAxis.Enable						:= stParameters.bStrawCatcherON;
		fbGearInCatcherAxis.GearRatio					:= 1;
		fbGearInAxisZ.Enable							:= TRUE;
		fbGearInAxisZ.GearRatio							:= SEL(stParameters.bStrawCatcherON, 1.0, 0.0000000001);
		
		
			IF (fbGearInCatcherAxis.InGear OR NOT stParameters.bStrawCatcherON) AND fbGearInAxisZ.InGear AND (tonStrawCatcher1Close.Q (*AND tonStrawCatcher2Close.Q*)
					OR (bStrawCatcherOpen1 AND bStrawCatcherOpen2 AND bStrawCatcherOpen3 AND bStrawCatcherOpen4))  THEN
				IF stParameters.bStrawCatcherON THEN
					eRunningState						:= E_CapPreScrewer.eCatching;	
				ELSE
					eRunningState						:= E_CapPreScrewer.ePlacing;	
				END_IF					
			END_IF		

	
	//Sprawdzanie czy chwytaki zamknięte i opuszczenie chwytaków do dolnej pozycji
	E_CapPreScrewer.eCatching:
		fbVirtualAxis.fPosition							:= (stParameters.LrCheckStrawCatcherActuatorZPosition - stParameters.lrStrawInsertDistance);	//Pozycja sprawdzania cofnięcia krabów
		fbVirtualAxis.fVelocity							:= SEL(stParameters.lrCatcherSpeed > 1094.0, stParameters.lrCatcherSpeed, 1094.0 );       						
		bVirtualMove									:= TRUE;				
	
	IF (CatcherAxisRef.NcToPlc.ActPos + stParameters.lrCatcherHightSV) <= (stParameters.lrCartesianCatchZPosition - (stParameters.lrCapHight + 25.0)) THEN	//+25
		fbGearInAxisZ.GearRatio								:= 1;
	END_IF
	
	//IF (CatcherAxisRef.NcToPlc.ActPos + stParameters.lrCatcherHightSV) <= (stParameters.lrCartesianCatchZPosition-(stParameters.lrCapHight)) THEN
	//	fbGearInAxisZ.GearRatio							:= 1;
	//END_IF
	
			//Otwórz chwytaki słomek
		IF CartesianZAxisRef.NcToPlc.ActPos <= stParameters.lrStrawCatcherZPosition THEN					
			bStrawCatchersOpen							:= TRUE;
			bStrawCatchersClose							:= FALSE;
			
				IF tonStrawCatcher1Open.Q AND tonStrawCatcher2Open.Q AND tonStrawCatcher3Open.Q AND tonStrawCatcher4Open.Q THEN																				
					//Cofnij chwytaki słomek
					bStrawCatcherActuatorIn				:= TRUE;
					bStrawCatcherActuatorOut			:= FALSE;				
				END_IF	
			
		END_IF		
		
		
		// 10mm stały offset - wysokość nad butelką
		//IF (CatcherAxisRef.NcToPlc.ActPos <= 1.0) OR (CatcherAxisRef.NcToPlc.ActPos <= ((stParameters.lrBottleHight) - stParameters.lrCatcherHightSV-20.0)) THEN	//20
		IF (CatcherAxisRef.NcToPlc.ActPos <= 1.0) OR (CatcherAxisRef.NcToPlc.ActPos + 32 <= ((stParameters.lrBottleHight + 10.0) - stParameters.lrCatcherHightSV)) THEN		
			fbGearInCatcherAxis.GearRatio				:= 0.0000000001;
				
				IF bStrawCatcherIn THEN
					fbGearInCatcherAxis.GearRatio		:= 0.0000000001;
					bVirtualMove						:= FALSE;	
					bStepButton							:= FALSE;
					eRunningState						:= E_CapPreScrewer.ePlacing;
				END_IF		
			
		END_IF
	


	
	//Czekaj aż chwytak słomek dojedzie do dołu i zacznij ruch osi pionowej Z
	E_CapPreScrewer.ePlacing:		
		IF stParameters.lrScrewFinding > 0 THEN
			eRunningState								:= E_CapPreScrewer.eFinding;
		ELSE
			lrPreScrewerAxisSavedPosition				:= PreScrewerAxisRef.NcToPlc.ActPos;	//zapisywanie pozycji przed zakrecaniem		
			fbVirtualAxis.fPosition						:= SEL(stParameters.bStrawCatcherON, stParameters.lrPlaceZPosition, stParameters.lrPlaceZPosition - stParameters.lrStrawInsertDistance);
			fbVirtualAxis.fVelocity						:= SEL(stParameters.lrCatcherSpeed > 1094.0, stParameters.lrCatcherSpeed, 1094.0 );    
			bVirtualMove								:= TRUE;
			
			eRunningState								:= E_CapPreScrewer.ePreScrewing;
		END_IF
	
	E_CapPreScrewer.eFinding:
		fbVirtualAxis.fPosition							:= SEL(stParameters.bStrawCatcherON, stParameters.lrScrewerStartZPosition, stParameters.lrScrewerStartZPosition-stParameters.lrStrawInsertDistance);
		fbVirtualAxis.fVelocity							:= SEL(stParameters.lrCatcherSpeed > 1094.0, stParameters.lrCatcherSpeed, 1094.0 );
		fbVirtualAxis.fAcceleration						:= stParameters.lrCatcherAcceleration; 
		fbVirtualAxis.fDeceleration						:= stParameters.lrCatcherAcceleration; 
		fbVirtualAxis.fJerk								:= stParameters.lrCatcherJerk;        		
			                                            
		bVirtualMove									:= TRUE;
		                                                
			IF ABS(fbVirtualAxis.Axis.NcToPlc.ActPos - fbVirtualAxis.fPosition) <= 0.5 THEN 

             
				bCapSucker[1]								:= FALSE;
				bCapSucker[2]								:= FALSE;
				bCapSucker[3]								:= FALSE;
				bCapSucker[4]								:= FALSE;
    	                                                
				mcPreScrewerMoveRelative.Distance		:= stParameters.lrScrewFinding * -1.0;
				mcPreScrewerMoveRelative.Acceleration	:= stParameters.lrScrewAcceleration;
				mcPreScrewerMoveRelative.Deceleration	:= stParameters.lrScrewAcceleration;
				mcPreScrewerMoveRelative.Velocity		:= stParameters.lrScrewSpeed;
				mcPreScrewerMoveRelative.Execute		:= TRUE;
			END_IF
			
					IF mcPreScrewerMoveRelative.Done OR ABS(PreScrewerAxisRef.NcToPlc.PosDiff) > 60.0 OR mcPreScrewerMoveRelative.Error THEN
						bVirtualMove							:= FALSE;
						mcPreScrewerMoveRelative.Execute		:= FALSE;
						eRunningState							:= E_CapPreScrewer.eScrewing;
					END_IF	
	
	E_CapPreScrewer.ePreScrewing:

	IF fbVirtualAxis.Axis.Status.Moving THEN
		bVirtualMove											:= FALSE;
		eRunningState											:= E_CapPreScrewer.eScrewing;
	END_IF
	
	
	E_CapPreScrewer.eScrewing:
		
				//8mm przed zakręcaniem synchronizuję prędkościowo posuw kartezjana
			IF CartesianZAxisRef.NcToPlc.ActPos <= stParameters.lrScrewerStartZPosition + 20 THEN	//+8
				
				
				fbVirtualAxis.fPosition					:= SEL(stParameters.bStrawCatcherON, stParameters.lrPlaceZPosition, stParameters.lrPlaceZPosition - stParameters.lrStrawInsertDistance);
				fbVirtualAxis.fVelocity					:= stParameters.lrPickerSpeedWhenScrewer;   
				fbVirtualAxis.fAcceleration				:= 100_000_000.0;
				fbVirtualAxis.fDeceleration				:= 100_000_000.0;
				fbVirtualAxis.fJerk						:= 100_000_000;//100_000_000_000;       
				bVirtualMove							:= TRUE;
			
						//1.0mm przed pozycją zakręcania załączam obrót
					IF CartesianZAxisRef.NcToPlc.ActPos <= stParameters.lrScrewerStartZPosition + 2.5 OR stVirtualMove_Out.Done THEN	
						lrPreScrewerAxisSavedPosition			:= PreScrewerAxisRef.NcToPlc.ActPos;	//zapisywanie pozycji przed zakrecaniem	potrzebna dla opcji otwierania chwytaków butelek	
						bCapSucker[1]							:= FALSE;
						bCapSucker[2]							:= FALSE;
						bCapSucker[3]							:= FALSE;
						bCapSucker[4]							:= FALSE;
						mcPreScrewerMoveRelative.Execute		:= TRUE;
						mcPreScrewerMoveRelative.Distance		:= stParameters.lrScrewDistance;
						mcPreScrewerMoveRelative.Acceleration	:= stParameters.lrScrewAcceleration;
						mcPreScrewerMoveRelative.Deceleration	:= stParameters.lrScrewAcceleration;
						mcPreScrewerMoveRelative.Velocity		:= stParameters.lrScrewSpeed;	
						eRunningState							:= E_CapPreScrewer.eFinished;	
					END_IF	
			END_IF
	
	//Kończenie cyklu zakręcania - otwarcie chwytaka
	E_CapPreScrewer.eFinished:		
					//otwórz centrowniki butelek
		//IF (GVL_Recipe.bCapSorterPreScrewerCatchAngleOpenEnaShow AND
		//	ABS(PreScrewerAxisRef.NcToPlc.ActPos - lrPreScrewerAxisSavedPosition) >= GVL_Recipe.lrCapSorterPreScrewerCatchAngleOpenSV) THEN
		//	bBottleCatcherCatchTemp					:= FALSE;
		//END_IF
	
		IF PreScrewerAxisRef.NcToPlc.PosDiff > 100.0 OR (mcPreScrewerMoveRelative.Done AND (stVirtualMove_Out.Done OR stVirtualMove2_Out.Done)) THEN
//			bBottleCatcherCatchTemp							:= FALSE;
			bCapCatcher1									:= FALSE;
		 	bCapCatcher2									:= FALSE;
		 	bCapCatcher3									:= FALSE;
		 	bCapCatcher4									:= FALSE;
			mcPreScrewerMoveRelative.Execute				:= FALSE;
			bVirtualMove									:= FALSE;
			
				IF fbVirtualAxis.Axis.Status.Moving THEN
					fbVirtualAxis.Halt(bExecute := TRUE);
				ELSIF PreScrewerAxisRef.Status.Moving THEN
					mcPreScrewerStop.Execute	:= TRUE;					
				ELSE
					mcPreScrewerStop.Execute	:= FALSE;
					fbVirtualAxis.Halt(bExecute := FALSE);
					fbGearInCatcherAxis.Enable				:= FALSE;
					fbGearInAxisZ.Enable					:= FALSE;
					eRunningState							:= E_CapPreScrewer.eGearOut;
				END_IF	
		END_IF
		
	E_CapPreScrewer.eGearOut:
		fbGearOutAxisZ.Execute								:= TRUE;
		fbGearOutCatcherAxis.Execute						:= TRUE;
	
			IF NOT CartesianZAxisRef.Status.Coupled AND NOT CatcherAxisRef.Status.Coupled THEN
				fbGearOutAxisZ.Execute						:= FALSE;
				fbGearOutCatcherAxis.Execute				:= FALSE;
				eRunningState								:= E_CapPreScrewer.eReturning1;
			END_IF
	
	//Powrót na górną pozycję
	E_CapPreScrewer.eReturning1:
	
		tonWaitInPlacePos.IN						:= TRUE;
		mcPreScrewerStop.Execute					:= TRUE;
		bCapCatcher1								:= FALSE;
		bCapCatcher2								:= FALSE;
		bCapCatcher3								:= FALSE;
		bCapCatcher4								:= FALSE;
		
		
		IF tonWaitInPlacePos.Q AND NOT PreScrewerAxisRef.Status.Moving THEN
			

		
			tonWaitInPlacePos.IN					:= FALSE;
//			bBottleCatcherCatchTemp					:= FALSE;		
			mcPreScrewerStop.Execute				:= FALSE;
			mcCartesianZMoveAbsolute.Execute		:= TRUE;
			mcCartesianZMoveAbsolute.Position		:= stParameters.lrTopZPosition;
			mcCartesianZMoveAbsolute.Acceleration	:= SEL(GVL_Recipe.iCapSorterProductType = 0 ,stParameters.lrPickerAcceleration , 150.0);
//			mcCartesianZMoveAbsolute.Acceleration	:= stParameters.lrPickerAcceleration;
			mcCartesianZMoveAbsolute.Deceleration	:= stParameters.lrPickerAcceleration;
			mcCartesianZMoveAbsolute.Velocity		:= stParameters.lrPickerSpeed;
			
			IF mcCartesianZMoveAbsolute.Busy THEN
				bCapBlow1								:= TRUE;
        		bCapBlow2								:= TRUE;
        		bCapBlow3								:= TRUE;
        		bCapBlow4								:= TRUE;	

					IF CartesianZAxisRef.NcToPlc.ActPos >= stParameters.lrScrewerStartZPosition	THEN
						bCapsBlowON								:= TRUE;
						mcCartesianZMoveAbsolute.Execute		:= FALSE;
						eRunningState							:= E_CapPreScrewer.eReturning2;
					END_IF		                                   
			END_IF
			
		END_IF
		

		
	//Powrót po osi X	
	E_CapPreScrewer.eReturning2:
		bBottleCatcherCatchTemp					:= FALSE;

		
		
		IF CartesianZAxisRef.NcToPlc.ActPos > stParameters.lrScrewerStartZPosition + 15.0 THEN
			mcCartesianZMoveAbsolute2.Execute		:= TRUE;
			mcCartesianZMoveAbsolute2.Position		:= stParameters.lrTopZPosition;
			mcCartesianZMoveAbsolute2.Acceleration	:= stParameters.lrPickerAcceleration;
			mcCartesianZMoveAbsolute2.Deceleration	:= stParameters.lrPickerAcceleration;
			mcCartesianZMoveAbsolute2.Velocity		:= stParameters.lrPickerSpeed;			
		END_IF
	
		IF (CartesianZAxisRef.NcToPlc.ActPos > stParameters.lrTopZPosition - stParameters.lrBendingDistance) OR
			mcCartesianZMoveAbsolute.Done THEN
			mcCatcherMoveAbsolute.Execute			:= TRUE;		
			mcCatcherMoveAbsolute.Position			:= stParameters.lrCatcherCatchingPosition;
			mcCatcherMoveAbsolute.Acceleration		:= stParameters.lrCatcherAcceleration;
			mcCatcherMoveAbsolute.Deceleration		:= stParameters.lrCatcherAcceleration;
			mcCatcherMoveAbsolute.Velocity			:= stParameters.lrCatcherSpeed;

//SEL(P190_CapFeeder.stMover2Status.bInPlacePosition, GVL_Recipe.lrCapSorterPreScrewerPickXMover1PositionShow, GVL_Recipe.lrCapSorterPreScrewerPickXMover2PositionShow

			
			//Jedź osią poziomą X na pozycję pick
			mcCartesianYMoveAbsolute.Execute		:= TRUE;
			{warning 'Przerobić, dodać parametry obu pozycji wózków do struktury parametrów, FB_CapPreScrewer.Running --> 624'}
			mcCartesianYMoveAbsolute.Position		:= SEL(bMover1InPickPos, GVL_Recipe.lrCapSorterPreScrewerPickXMover1PositionShow, GVL_Recipe.lrCapSorterPreScrewerPickXMover2PositionShow);
			mcCartesianYMoveAbsolute.Acceleration	:= stParameters.lrPickerAcceleration;
			mcCartesianYMoveAbsolute.Deceleration	:= stParameters.lrPickerAcceleration;
			mcCartesianYMoveAbsolute.Velocity		:= stParameters.lrPickerSpeed;
			//Ustaw obracarkę do pozycji początkowej
			
			mcPreScrewerMoveRelative.Distance		:= -1 * DINT_TO_LREAL(LREAL_TO_DINT(PreScrewerAxisRef.NcToPlc.SetPos) MOD 360); 
			mcPreScrewerMoveRelative.Execute		:= mcPreScrewerMoveRelative.Distance<>0 AND NOT mcPreScrewerMoveRelative.Error;
			mcPreScrewerMoveRelative.Acceleration	:= stParameters.lrScrewAcceleration;
			mcPreScrewerMoveRelative.Deceleration	:= stParameters.lrScrewAcceleration;
			mcPreScrewerMoveRelative.Velocity		:= stParameters.lrScrewSpeed;
			
		END_IF
		IF CartesianZAxisRef.NcToPlc.ActPos > stParameters.lrPlaceZPosition + 20 THEN
			bPlaceDone								:= TRUE;
		END_IF
		IF (*bPlaceDone AND*) mcCartesianYMoveAbsolute.Done AND mcCartesianZMoveAbsolute2.Done AND
			 mcCatcherMoveAbsolute.Done AND NOT bCapBlow1 AND NOT bCapBlow2 AND NOT bCapBlow3 AND NOT bCapBlow4 THEN
				 IF mcPreScrewerMoveRelative.Distance=0 OR mcPreScrewerMoveRelative.Done THEN
					mcCartesianYMoveAbsolute.Execute		:= FALSE;
 					mcCartesianZMoveAbsolute.Execute		:= FALSE;
					mcCartesianZMoveAbsolute2.Execute		:= FALSE;
					mcCatcherMoveAbsolute.Execute			:= FALSE;
					mcPreScrewerMoveRelative.Execute		:= FALSE;
					eRunningState				:= E_CapPreScrewer.eDone;
				END_IF
		END_IF
		
		//Dodatkowy przedmuch ssawek
		(*IF (CartesianZAxisRef.NcToPlc.ActPos > (stParameters.lrPlaceZPosition + stParameters.lrHeightAdditionalBlow)) THEN
			bAdditionalBlow							S= NOT tonBlowOFF.IN;	
		
			IF NOT bAdditionalBlow THEN
				bCapsBlowON							R= tonBlowOFF.Q;
			END_IF

			bCapsBlowON								S= bAdditionalBlow;
			bCapBlow1 := bCapBlow2 := bCapBlow3 := bCapBlow4 := bAdditionalBlow;
		END_IF*)
			
	E_CapPreScrewer.eDone:
		mcPreScrewerStop.Execute				:= TRUE;
	
		IF mcPreScrewerStop.Done THEN
			mcPreScrewerStop.Execute			:= FALSE;
			bAdditionalBlow						:= FALSE;
			bCycleNotDone						:= FALSE;
			bCapsBlowON							:= FALSE;
			bPlaceDone							:= TRUE;
			bCycleDone							:= TRUE;
			eState								:= E_Station.eDone;
			eRunningState						:= E_CapPreScrewer.eReady;	
		END_IF	

	(*Cykl nie zakończony - przerwany - chyba nie potrzebny*)
	E_CapPreScrewer.eNotDone:
		bCapsBlowON							:= FALSE;
		eState								:= E_Station.eDone;
		eRunningState						:= E_CapPreScrewer.eReady;




END_CASE

tonCapCatcher(PT := T#60MS);
END_ACTION

ACTION RunningCam:

tonVacuumWatchdog(PT	:= stParameters.tTimeVacuumWatchdog);
bStopAllowed	:= eRunningState = E_CapPreScrewer.eReady OR eRunningState = E_CapPreScrewer.eVerticalDownToCatchPos;

//Otwieranie chwytaków
//bBottleCatcherCatchTemp		R= CartesianZAxisRef.NcToPlc.ActPos < stParameters.lrGripperOpenPosition;
GVL_VIS.bCapSorterPreScrewerBottleCatcherCatch	:= bBottleCatcherCatchTemp AND bCapSorterPreScrewerBottleCatcherEnableShow;
	
tonWaitInPlacePos(PT	:= stParameters.tWaitInPlacePos);
//tonWaitInPlacePos(PT 	:= T#200MS);
eLastRunningState	:= eRunningState;

CASE eRunningState OF

//====================================
	
	(*Oczekiwanie na wykonanie pojedynczego cyklu*)
	E_CapPreScrewer.eReady:

		
		IF NOT bCycleDone AND NOT bCycleNotDone THEN  
                                      	
			IF bRun THEN 
				fbVirtualAxis.fAcceleration				:= stParameters.lrPickerAcceleration;	//100_000_000.0;
				fbVirtualAxis.fDeceleration				:= stParameters.lrPickerAcceleration;	//100_000_000.0;
				fbVirtualAxis.fJerk						:= stParameters.lrPickerJerk;// 	1_000_000;//100_000_000_000;  

				iRejectCase					:= 0;
				bRejectDone					:= FALSE;
				bReject						:= FALSE;
				bTubeReject					:= FALSE;
				
				//Przygotuj do cyklu - otwórz chwytaki
				bCapCatcher1				:= FALSE;
				bCapCatcher2				:= FALSE;
				bCapCatcher3				:= FALSE;
				bCapCatcher4				:= FALSE;
	
				//Wyłącz ssawki
				bCapSucker[1]				:= FALSE;
				bCapSucker[2]				:= FALSE;
				bCapSucker[3]				:= FALSE;
				bCapSucker[4]				:= FALSE;
				//Wyłącz odmuchy
				bCapBlower1					:= FALSE;
				bCapBlower2					:= FALSE;
				bCapBlower3					:= FALSE;
				bCapBlower4					:= FALSE;
				bCapsBlowON					:= FALSE;
				//Otwórz chwytaki słomek
				bStrawCatchersOpen			:= TRUE;
				bStrawCatchersClose			:= FALSE;
				//Cofnij chwytaki słomek
				bStrawCatcherActuatorIn		:= TRUE;
				bStrawCatcherActuatorOut	:= FALSE;
				//Podjedź robotem i chwytakiem słomek w górę jak cofnięty chwytak słomek
				IF tonStrawCatcherIn.Q THEN	
										
					mcCartesianZMoveAbsolute.Execute		:= TRUE;		
					mcCartesianZMoveAbsolute.Position		:= stParameters.lrTopZPosition;
					mcCartesianZMoveAbsolute.Acceleration	:= stParameters.lrPickerAcceleration;
					mcCartesianZMoveAbsolute.Deceleration	:= stParameters.lrPickerAcceleration;
					mcCartesianZMoveAbsolute.Velocity		:= stParameters.lrPickerSpeed;
					
					mcCatcherMoveAbsolute.Execute			:= TRUE;		
					mcCatcherMoveAbsolute.Position			:= stParameters.lrCatcherCatchingPosition;
					mcCatcherMoveAbsolute.Acceleration		:= stParameters.lrCatcherAcceleration;
					mcCatcherMoveAbsolute.Deceleration		:= stParameters.lrCatcherAcceleration;
					mcCatcherMoveAbsolute.Velocity			:= stParameters.lrCatcherSpeed;
					
					//Następny krok
					eRunningState						:= E_CapPreScrewer.ePreparingToPick;
					bCycleNotDone						:= TRUE;
					
				END_IF
				//Reset komendy ruchu osi X
				mcCartesianYMoveAbsolute.Execute		:= FALSE;
				
			END_IF
		END_IF
			
	(*Czekam na pozycję Z w górze i ruszam osią poziomą X na pozycję pobierania i czekam na obie pozycje*)
	E_CapPreScrewer.ePreparingToPick:
		IF (CartesianZAxisRef.NcToPlc.ActPos > stParameters.lrTopZPosition - stParameters.lrBendingDistance) OR
			mcCartesianZMoveAbsolute.Done THEN
			//Jedź osią poziomą X na pozycję pick
			mcCartesianYMoveAbsolute.Execute		:= TRUE;
			mcCartesianYMoveAbsolute.Position		:= stParameters.lrPickYPosition;
			mcCartesianYMoveAbsolute.Acceleration	:= stParameters.lrPickerAcceleration;
			mcCartesianYMoveAbsolute.Deceleration	:= stParameters.lrPickerAcceleration;
			mcCartesianYMoveAbsolute.Velocity		:= stParameters.lrPickerSpeed;
			//Nakrętka pobrana z wózka nr.1
			bMover1InPickPos						:= SEL((stParameters.lrPickYPosition-GVL_Recipe.lrCapSorterPreScrewerPickXMover1PositionShow) <= 0.5, FALSE, TRUE);
			
			//Ustaw obracarkę w pozycji
			mcPreScrewerMoveRelative.Distance		:=  -1 * DINT_TO_LREAL((LREAL_TO_DINT(PreScrewerAxisRef.NcToPlc.SetPos)+diPreSCrewerHomePos) MOD 360);
			mcPreScrewerMoveRelative.Execute		:= mcPreScrewerMoveRelative.Distance<>0;
			mcPreScrewerMoveRelative.Acceleration	:= stParameters.lrScrewAcceleration;
			mcPreScrewerMoveRelative.Deceleration	:= stParameters.lrScrewAcceleration;
			mcPreScrewerMoveRelative.Velocity		:= stParameters.lrScrewSpeed;
		END_IF
		//Jak obie pozycje osiągnięte to wysuń chwytak słomek i następny krok
		IF mcCartesianYMoveAbsolute.Done AND mcCartesianZMoveAbsolute.Done AND mcCatcherMoveAbsolute.Done THEN
			IF mcPreScrewerMoveRelative.Done OR mcPreScrewerMoveRelative.Distance =0 THEN
				//Reset komendy ruchu osi
				mcCartesianYMoveAbsolute.Execute		:= FALSE;
				mcCartesianZMoveAbsolute.Execute		:= FALSE;
				mcPreScrewerMoveRelative.Execute		:= FALSE;
				mcCatcherMoveAbsolute.Execute			:= FALSE;
				//Wysuń chwytaki słomek jesli to potrzebuje recepta        
				bStrawCatcherActuatorIn					:= NOT stParameters.bStrawCatcherON;
				bStrawCatcherActuatorOut				:= stParameters.bStrawCatcherON;    
				//Następny krok
				eRunningState							:= E_CapPreScrewer.ePicking;
			END_IF
		END_IF
		
	
	(*Zjeżdzam na osią pionową Z na pozycję chwytania i załączam ssawki*)		
	E_CapPreScrewer.ePicking:
		//Podjedź robotem w górę	
		mcCartesianZMoveAbsolute.Execute			:= TRUE;		
		mcCartesianZMoveAbsolute.Position			:= stParameters.lrPickZPosition;
		mcCartesianZMoveAbsolute.Acceleration		:= stParameters.lrPickerAcceleration;
		mcCartesianZMoveAbsolute.Deceleration		:= stParameters.lrPickerAcceleration;
		mcCartesianZMoveAbsolute.Velocity			:= stParameters.lrPickerSpeed;
		//Czekam na wykonanie ruchu
		IF mcCartesianZMoveAbsolute.Done THEN
			//Reset komendy ruchu osi
			mcCartesianZMoveAbsolute.Execute		:= FALSE;
			
			//Zeruje rejestry oraz załączanie ssawek
			 FOR i:=1 TO 4 DO
				 bCapSucker[i]						:= stParameters.bPickerActiv[i]; 
				 aCapPresence[i] 					:= FALSE;
			 END_FOR
	
			//Następny krok
			eRunningState							:= E_CapPreScrewer.eVacumCheckPart1;
		END_IF
	
	(*Sprawdzam czy zassane i jazda w górę*)	
	E_CapPreScrewer.eVacumCheckPart1:
		
		tonVacuumWatchdog.IN						:= TRUE;
		
		IF tonSuckedOk[1].Q = stParameters.bPickerActiv[1] AND tonSuckedOk[2].Q = stParameters.bPickerActiv[2]
			AND tonSuckedOk[3].Q = stParameters.bPickerActiv[3] AND tonSuckedOk[4].Q = stParameters.bPickerActiv[4] THEN
			tonVacuumWatchdog.IN					:= FALSE;
		
				FOR i:=1 TO 4 DO
					IF stParameters.bPickerActiv[i] AND stParameters.bStrawCatcherON AND NOT stMoverStatus.stSlotStatus[i].bTubePresent THEN
						bReject								:= TRUE;
						bTubeReject							:= TRUE;
						lrAxisZ_RejectOffset				:= 0.0;
					END_IF

					IF bMover1InPlacePos THEN
						diMover1VacuumRetry[i]		:= 0;
					ELSE
						diMover2VacuumRetry[i]		:= 0;
					END_IF	
				END_FOR 
				
			eRunningState 							:= E_CapPreScrewer.eVacumCheckPart2;
	
		ELSIF tonVacuumWatchdog.Q THEN
		
			FOR i:=1 TO 4 DO
				bCapSucker[i]							:= tonSuckedOk[i].Q;
				
				//robimy odrzut jeżeli zostanie wykryto brak słomki
				IF stParameters.bPickerActiv[i] AND stParameters.bStrawCatcherON AND NOT stMoverStatus.stSlotStatus[i].bTubePresent THEN
					bReject								:= TRUE;
					bTubeReject							:= TRUE;
					lrAxisZ_RejectOffset				:= 0.0;
				END_IF
				
						//Detekcja niepobranej nasadki --> odrzut aktywowany opcjonalnie z receptury
					IF stParameters.bPickerActiv[i] AND NOT tonSuckedOk[i].Q AND NOT stParameters.bVacuumDeactivate THEN
						bReject							:= SEL(stParameters.bRejectON, bReject, TRUE);
						lrAxisZ_RejectOffset			:= SEL(stParameters.bRejectON, lrAxisZ_RejectOffset, 13.0);	//offset dodatkowego zjazdu kartezjanem 
						
						IF bMover1InPlacePos THEN
							diMover1VacuumRetry[i]		:= diMover1VacuumRetry[i] + 1;
						ELSE	
							diMover2VacuumRetry[i]		:= diMover2VacuumRetry[i] + 1;
						END_IF
					ELSIF tonSuckedOk[i].Q OR stParameters.bVacuumDeactivate THEN
						IF 	bMover1InPlacePos THEN
							diMover1VacuumRetry[i]		:= 0;
						ELSE
							diMover2VacuumRetry[i]		:= 0;
						END_IF	
					END_IF	
	    	
			END_FOR
				tonVacuumWatchdog.IN					:= FALSE;
				eRunningState 							:= E_CapPreScrewer.eVacumCheckPart2;
	
		END_IF
		
		
	E_CapPreScrewer.eVacumCheckPart2:	
			
		//Jezeli nie jest przyssana zadna nasadka to pdjezdzamy na poz. ready oraz wystawiamy flage bMissingCaps
		IF bReject THEN
			Reject();
				IF bRejectDone THEN				
					eRunningState						:= E_CapPreScrewer.eReady;	
				END_IF		
		ELSIF NOT tonSuckedOk[1].Q AND NOT tonSuckedOk[2].Q AND NOT tonSuckedOk[3].Q AND NOT tonSuckedOk[4].Q THEN
			bCapSucker[1]							:= FALSE;
			bCapSucker[2]							:= False;
			bCapSucker[3]							:= False;
		    bCapSucker[4]							:= False;	
			mcCartesianZMoveAbsolute.Execute		:= TRUE;		
			mcCartesianZMoveAbsolute.Position		:= stParameters.lrTopZPosition;
			mcCartesianZMoveAbsolute.Acceleration	:= stParameters.lrPickerAcceleration;
			mcCartesianZMoveAbsolute.Deceleration	:= stParameters.lrPickerAcceleration;
			mcCartesianZMoveAbsolute.Velocity		:= stParameters.lrPickerSpeed;
			
			IF mcCartesianZMoveAbsolute.Done THEN
				bMissingCaps						:= TRUE;
				bCycleDone;
				mcCartesianZMoveAbsolute.Execute	:= FALSE;
				eRunningState						:= E_CapPreScrewer.eReady;	
			END_IF
			
		ELSE
			mcCartesianZMoveAbsolute.Execute		:= NOT stParameters.bVacuumDeactivate;		
			mcCartesianZMoveAbsolute.Position		:= stParameters.lrTopZPosition;
			mcCartesianZMoveAbsolute.Acceleration	:= SEL(GVL_Recipe.iCapSorterProductType = 0 ,stParameters.lrPickerAcceleration , 150.0);//stParameters.lrPickerAcceleration;
//			mcCartesianZMoveAbsolute.Acceleration	:= stParameters.lrPickerAcceleration;
			mcCartesianZMoveAbsolute.Deceleration	:= stParameters.lrPickerAcceleration;
			mcCartesianZMoveAbsolute.Velocity		:= stParameters.lrPickerSpeed;
			tonCapCatcher.IN						:= FALSE;
			
			IF mcCartesianZMoveAbsolute.Busy OR stParameters.bVacuumDeactivate THEN
				mcCartesianZMoveAbsolute.Execute		:= FALSE;
				eRunningState 							:= E_CapPreScrewer.eTransferingVertical; 
			END_IF
			
        
		END_IF		
			
			//przepisuje do rejestrów nakretki które kartezjan pobrał
			aCapPresence[1] := bCapSucker[1];
			aCapPresence[2] := bCapSucker[2];
			aCapPresence[3] := bCapSucker[3];
			aCapPresence[4] := bCapSucker[4];						

		
		
	(*Jazda w górę, zamknięcie łapek i załączenie jazdy w bok*)	
	E_CapPreScrewer.eTransferingVertical:
		
		IF NOT bCapSucker[1] OR NOT bCapSucker[2] OR NOT bCapSucker[3] OR NOT bCapSucker[4] THEN
            bCapBlow1						:= NOT bCapSucker[1];
            bCapBlow2						:= NOT bCapSucker[2];
            bCapBlow3						:= NOT bCapSucker[3];
            bCapBlow4						:= NOT bCapSucker[4];						
			bCapsBlowON						:= TRUE;
		END_IF
		
		//Kleją się kulki 
		IF NOT stParameters.bVacuumDeactivate THEN					
			IF CartesianZAxisRef.NcToPlc.ActPos > stParameters.lrPickZPosition + 10.0 THEN
				mcCartesianZMoveAbsolute2.Execute		:= NOT stParameters.bVacuumDeactivate;		
				mcCartesianZMoveAbsolute2.Position		:= SEL(stParameters.lrCartesianCatchZPosition > stParameters.lrTopZPosition, stParameters.lrTopZPosition, stParameters.lrCartesianCatchZPosition);
				mcCartesianZMoveAbsolute2.Acceleration	:= stParameters.lrPickerAcceleration;
				mcCartesianZMoveAbsolute2.Deceleration	:= stParameters.lrPickerAcceleration;
				mcCartesianZMoveAbsolute2.Velocity		:= stParameters.lrPickerSpeed;
			END_IF
		END_IF


		IF CartesianZAxisRef.NcToPlc.ActPos > stParameters.lrCapCatcherZPosition  THEN //OR (CartesianZAxisRef.Status.Moving)
			bCapCatcher1							:= TRUE;
			bCapCatcher2							:= true;
			bCapCatcher3							:= true;
			bCapCatcher4							:= true;
			tonCapCatcher.IN						:= stParameters.bVacuumDeactivate;
		END_IF	
		
		mcCartesianZMoveAbsolute.Execute		:= tonCapCatcher.Q;	
		
		//Dodać sprawdzenie czy gotowy chwytak słomek !!!!!
		//Sprawdzenie pozycji osi pionowej Z i czy wysunięty siłownik chwytaka słomek
		IF ((CartesianZAxisRef.NcToPlc.ActPos > stParameters.lrTopZPosition - stParameters.lrBendingDistance) OR
			mcCartesianZMoveAbsolute.Done) AND (tonStrawCatcherOut.Q OR NOT stParameters.bStrawCatcherON) THEN
			//Jedź osią poziomą X na pozycję pick
				mcCartesianZMoveAbsolute2.Execute		:= FALSE;
				bCapsBlowON								:= FALSE;
				eRunningState 							:= E_CapPreScrewer.eTransferingHorizontal;
				tonCapCatcher.IN						:= FALSE;
		END_IF
	
	(*Przejazd w poziomie*)	
	E_CapPreScrewer.eTransferingHorizontal:	
	
			bCapCatcher1							:= TRUE;//bCapSucker1;
			bCapCatcher2							:= TRUE;//bCapSucker2;
			bCapCatcher3							:= TRUE;//bCapSucker3;
			bCapCatcher4							:= TRUE;//bCapSucker4;
	
		mcCartesianYMoveAbsolute.Position			:= stParameters.lrPlaceYPosition;
		mcCartesianYMoveAbsolute.Acceleration		:= stParameters.lrPickerAcceleration;
		mcCartesianYMoveAbsolute.Deceleration		:= stParameters.lrPickerAcceleration;
		mcCartesianYMoveAbsolute.Velocity			:= stParameters.lrPickerSpeed;
		mcCartesianYMoveAbsolute.Execute			:= TRUE;
		
		IF (CartesianYAxisRef.NcToPlc.ActPos > 200.0 (*stParameters.lrPlaceYPosition - stParameters.lrBendingDistance*)) OR
			mcCartesianYMoveAbsolute.Done AND NOT mcCartesianZMoveAbsolute.Execute THEN			

			//Podjedź robotem w dól	
			mcCartesianZMoveAbsolute.Execute			:= TRUE;		
			mcCartesianZMoveAbsolute.Position			:= stParameters.lrCartesianCatchZPosition;
			mcCartesianZMoveAbsolute.Acceleration		:= stParameters.lrPickerAcceleration;
			mcCartesianZMoveAbsolute.Deceleration		:= stParameters.lrPickerAcceleration;
			mcCartesianZMoveAbsolute.Velocity			:= stParameters.lrPickerSpeed;
		END_IF
		
		//Jak obie pozycje osiągnięte 
		IF mcCartesianZMoveAbsolute.Done THEN
			mcCartesianZMoveAbsolute.Execute		:= FALSE;
		END_IF
			
		//Jak ak obie pozycje osiągnięte to zamykamy chwytaki i następny krok
		IF stParameters.bStrawCatcherON AND CartesianYAxisRef.NcToPlc.ActPos >= stParameters.lrPlaceYPosition THEN
			//Zamknij chwytaki słomek
			bStrawCatchersOpen						:= FALSE;
			bStrawCatchersClose						:= TRUE;	
		END_IF
		
			
		IF  mcCartesianYMoveAbsolute.Done AND mcCartesianZMoveAbsolute.Done THEN			
				//Ustaw pozycję wirtualnej osi tak samo jak na osi Z
			fbVirtualAxis.fPosition						:=  CartesianZAxisRef.NcToPlc.ActPos;
			fbVirtualAxis.SetPosAbsClearLag(bExecute	:= TRUE);
				
				IF fbVirtualAxis.pSetPos.Busy THEN
						//Reset komendy ruchu osi
					mcCartesianYMoveAbsolute.Execute	:= FALSE;
					mcCartesianZMoveAbsolute.Execute	:= FALSE;
					//Następny krok
					eRunningState						:= E_CapPreScrewer.eVerticalDownToCatchPos;	
				END_IF
		END_IF		
		
	(*Przejazd w dól do pozycji chwytanija rurki*)		
	E_CapPreScrewer.eVerticalDownToCatchPos:
		fbVirtualAxis.SetPosAbsClearLag(bExecute				:= FALSE);
		
		//Jak ak obie pozycje osiągnięte to zamykamy chwytaki i następny krok
		IF stParameters.bStrawCatcherON THEN
			//Zamknij chwytaki słomek
			bStrawCatchersOpen					:= FALSE;
			bStrawCatchersClose					:= TRUE;	
			//Generowanie krzywki
			CamCalculation();
			fbCamTableSelectCatcher.Execute		:= TRUE;	
			fbCamTableSelectAxisZ.Execute		:= TRUE;
		END_IF
				
			IF tonPlacePermission.Q AND (NOT stParameters.bStrawCatcherON OR (tonStrawCatcher1Close.Q AND fbCamTableSelectCatcher.Done AND fbCamTableSelectAxisZ.Done)) THEN	
					fbCamTableSelectCatcher.Execute		:= FALSE;
				   	fbCamTableSelectAxisZ.Execute		:= FALSE;
					bCapCatcher1						:= TRUE;
					bCapCatcher2						:= TRUE;
					bCapCatcher3						:= TRUE;
					bCapCatcher4						:= TRUE;						
					eRunningState						:= E_CapPreScrewer.eAxisGearIn;
			END_IF
		
	
	E_CapPreScrewer.eAxisGearIn:
	
		IF stParameters.bStrawCatcherON THEN
			fbCamInAxisZ.Execute						:= TRUE;
			fbCamInAxisCatcher.Execute					:= TRUE;
			
				IF fbCamInAxisZ.InSync AND fbCamInAxisCatcher.InSync THEN
					fbCamInAxisZ.Execute				:= FALSE;
					fbCamInAxisCatcher.Execute			:= FALSE;
				
				
					eRunningState					:= E_CapPreScrewer.ePositionOverBottle;	
					fbVirtualAxis.fPosition			:= (stParameters.LrCheckStrawCatcherActuatorZPosition - arrTableAxisZ[1,0]);	
					fbVirtualAxis.fVelocity			:= SEL(stParameters.lrCatcherSpeed > 1094.0, stParameters.lrCatcherSpeed, 1094.0 ); 
					bVirtualMove					:= TRUE;	
					eRunningState					:= E_CapPreScrewer.ePositionOverBottle;	
				END_IF	
		ELSE                            
			mcCartesianZMoveAbsolute.Execute		:= TRUE;		
			mcCartesianZMoveAbsolute.Position		:= stParameters.lrScrewerStartZPosition;
			mcCartesianZMoveAbsolute.Acceleration	:= stParameters.lrPickerAcceleration;
			mcCartesianZMoveAbsolute.Deceleration	:= stParameters.lrPickerAcceleration;
			mcCartesianZMoveAbsolute.Velocity		:= stParameters.lrPickerSpeed;
			eRunningState							:= E_CapPreScrewer.ePlacing;	
		END_IF	

	
	
	E_CapPreScrewer.ePositionOverBottle:		      			
		IF fbVirtualAxis.Axis.Status.Moving THEN
			bVirtualMove							:= FALSE;
			eRunningState							:= E_CapPreScrewer.eCatching;	
		END_IF
	
	
	//Sprawdzanie czy chwytaki zamknięte i opuszczenie chwytaków do dolnej pozycji
	E_CapPreScrewer.eCatching:
	
			//Otwórz chwytaki słomek
		IF CartesianZAxisRef.NcToPlc.ActPos <= stParameters.lrStrawCatcherZPosition THEN		
			bStrawCatchersOpen							:= TRUE;
			bStrawCatchersClose							:= FALSE;
			
				IF tonStrawCatcher1Open.Q AND tonStrawCatcher2Open.Q AND tonStrawCatcher3Open.Q AND tonStrawCatcher4Open.Q THEN																				
					//Cofnij chwytaki słomek
					bStrawCatcherActuatorIn				:= TRUE;
					bStrawCatcherActuatorOut			:= FALSE;				
				END_IF	
		END_IF		
						
				IF bStrawCatcherIn THEN	
					eRunningState						:= E_CapPreScrewer.ePlacing;
					fbVirtualAxis.fPosition				:= stParameters.lrScrewerStartZPosition - arrTableAxisZ[1,0];
					fbVirtualAxis.fVelocity				:= SEL(stParameters.lrCatcherSpeed > 1094.0, stParameters.lrCatcherSpeed, 1094.0 );    
					bVirtualMove						:= TRUE;
				END_IF		
			
		//END_IF
	


	
	//Czekaj aż chwytak słomek dojedzie do dołu i zacznij ruch osi pionowej Z
	E_CapPreScrewer.ePlacing:		
	
		IF stParameters.lrScrewFinding > 0 THEN
			eRunningState								:= E_CapPreScrewer.eFinding;
		ELSE
			eRunningState								:= E_CapPreScrewer.ePreScrewing;
		END_IF
	
	E_CapPreScrewer.eFinding:		                                                
			IF stParameters.bStrawCatcherON THEN
				IF ABS(fbVirtualAxis.Axis.NcToPlc.ActPos - fbVirtualAxis.fPosition) <= 3.0 THEN              
					bCapSucker[1]								:= FALSE;
					bCapSucker[2]								:= FALSE;
					bCapSucker[3]								:= FALSE;
					bCapSucker[4]								:= FALSE;
    	        	                                        
					mcPreScrewerMoveRelative.Distance		:= stParameters.lrScrewFinding * -1.0;
					mcPreScrewerMoveRelative.Acceleration	:= stParameters.lrScrewAcceleration;
					mcPreScrewerMoveRelative.Deceleration	:= stParameters.lrScrewAcceleration;
					mcPreScrewerMoveRelative.Velocity		:= stParameters.lrScrewSpeed;
					mcPreScrewerMoveRelative.Execute		:= TRUE;
				END_IF	
			ELSE	
				IF ABS(CartesianZAxisRef.NcToPlc.ActPos - mcCartesianZMoveAbsolute.Position) <= 3.0 THEN 
					bCapSucker[1]								:= FALSE;
					bCapSucker[2]								:= FALSE;
					bCapSucker[3]								:= FALSE;
					bCapSucker[4]								:= FALSE;
    	        	                                        
					mcPreScrewerMoveRelative.Distance		:= stParameters.lrScrewFinding * -1.0;
					mcPreScrewerMoveRelative.Acceleration	:= stParameters.lrScrewAcceleration;
					mcPreScrewerMoveRelative.Deceleration	:= stParameters.lrScrewAcceleration;
					mcPreScrewerMoveRelative.Velocity		:= stParameters.lrScrewSpeed;
					mcPreScrewerMoveRelative.Execute		:= TRUE;
				END_IF
			END_IF
			
					IF mcPreScrewerMoveRelative.Done OR ABS(PreScrewerAxisRef.NcToPlc.PosDiff) > 60.0 OR mcPreScrewerMoveRelative.Error THEN
						bVirtualMove							:= FALSE;
						mcPreScrewerMoveRelative.Execute		:= FALSE;
						eRunningState							:= E_CapPreScrewer.ePreScrewing;
					END_IF	
	
	E_CapPreScrewer.ePreScrewing:

		IF stParameters.bStrawCatcherON THEN
			IF ABS(fbVirtualAxis.Axis.NcToPlc.ActPos - fbVirtualAxis.fPosition)<=0.1 THEN
				bVirtualMove											:= FALSE;
				
				IF NOT	CartesianZAxisRef.Status.SynchronizedMotion AND NOT CartesianZAxisRef.Status.Moving THEN
					eRunningState				:= E_CapPreScrewer.eScrewing;
					mcCartesianZStop.Execute	:= FALSE;
					fbCamOutAxisZ.Execute		:= FALSE;
				ELSE
					fbCamOutAxisZ.Execute		:= TRUE;
					mcCartesianZStop.Execute	:= CartesianZAxisRef.Status.Moving;
				END_IF	
			END_IF
		ELSE
			IF mcCartesianZMoveAbsolute.Done THEN
				eRunningState						:= E_CapPreScrewer.eScrewing;
				mcCartesianZMoveAbsolute.Execute	:= FALSE;
			END_IF	
		END_IF
		
	
	
	E_CapPreScrewer.eScrewing:
	
			fbGearInAxisZ_Screwer.Execute			:= NOT CartesianZAxisRef.Status.Coupled AND NOT mcCartesianZStop.Busy;
			fbGearInAxisZ_Screwer.RatioNumerator 	:= (GVL_Recipe.lrCapSorterPreScrewerThreadPitchShow	* GVL_Recipe.lrCapSorterPreScrewerMultipleStartThreadShow * (-1));
			fbGearInAxisZ_Screwer.RatioDenominator	:= 360;
		
			IF CartesianZAxisRef.Status.Coupled THEN
						mcPreScrewerMoveRelative.Execute		:= TRUE;
						mcPreScrewerMoveRelative.Distance		:= stParameters.lrScrewDistance;
						mcPreScrewerMoveRelative.Acceleration	:= stParameters.lrScrewAcceleration;
						mcPreScrewerMoveRelative.Deceleration	:= stParameters.lrScrewAcceleration;
						mcPreScrewerMoveRelative.Velocity		:= stParameters.lrScrewSpeed;	
						eRunningState							:= E_CapPreScrewer.eFinished;	
			END_IF
	
	//Kończenie cyklu zakręcania - otwarcie chwytaka
	E_CapPreScrewer.eFinished:		
	
		IF PreScrewerAxisRef.NcToPlc.PosDiff > 100.0 OR mcPreScrewerMoveRelative.Done THEN
//			bBottleCatcherCatchTemp							:= FALSE;	
			bCapCatcher1									:= FALSE;
		 	bCapCatcher2									:= FALSE;
		 	bCapCatcher3									:= FALSE;
		 	bCapCatcher4									:= FALSE;
			mcPreScrewerMoveRelative.Execute				:= FALSE;
			bVirtualMove									:= FALSE;
			bCapBlow1										:= stParameters.bPickerActiv[1];
            bCapBlow2										:= stParameters.bPickerActiv[2];
            bCapBlow3										:= stParameters.bPickerActiv[3];
            bCapBlow4										:= stParameters.bPickerActiv[4];
			bCapSucker[1]									:= FALSE;
			bCapSucker[2]									:= FALSE;
			bCapSucker[3]									:= FALSE;
			bCapSucker[4]									:= FALSE;								
			
				IF PreScrewerAxisRef.Status.Moving THEN
					mcPreScrewerStop.Execute				:=	 TRUE;					
				ELSE
					lrAxisZSavedPosition					:= CartesianZAxisRef.NcToPlc.ActPos;
					mcPreScrewerStop.Execute				:= FALSE;
					fbGearInCatcherAxis.Enable				:= FALSE;
					eRunningState							:= E_CapPreScrewer.eGearOut;
				END_IF	
		END_IF
		
	E_CapPreScrewer.eGearOut:
		fbGearOutAxisZ.Execute								:= TRUE;
		fbCamOutAxisCatcher.Execute							:= TRUE;
	
			IF NOT CartesianZAxisRef.Status.Coupled AND NOT CatcherAxisRef.Status.SynchronizedMotion THEN
				fbGearOutAxisZ.Execute						:= FALSE;
				fbCamOutAxisCatcher.Execute					:= FALSE;
				eRunningState								:= E_CapPreScrewer.eReturning1;
			END_IF
	
	//Powrót na górną pozycję
	E_CapPreScrewer.eReturning1:
	
		tonWaitInPlacePos.IN						:= TRUE;
		mcPreScrewerStop.Execute					:= TRUE;		

		IF tonWaitInPlacePos.Q THEN
			

		
			tonWaitInPlacePos.IN					:= FALSE;
//			bBottleCatcherCatchTemp					:= FALSE;		
			mcPreScrewerStop.Execute				:= FALSE;
			mcCartesianZMoveAbsolute.Execute		:= TRUE;
			mcCartesianZMoveAbsolute.Position		:= stParameters.lrTopZPosition;
			mcCartesianZMoveAbsolute.Acceleration	:= SEL(GVL_Recipe.iCapSorterProductType = 0 ,stParameters.lrPickerAcceleration , 150.0);
//			mcCartesianZMoveAbsolute.Acceleration	:= stParameters.lrPickerAcceleration;
			mcCartesianZMoveAbsolute.Deceleration	:= stParameters.lrPickerAcceleration;
			mcCartesianZMoveAbsolute.Velocity		:= stParameters.lrPickerSpeed;
			
			IF mcCartesianZMoveAbsolute.Busy THEN
				mcCartesianZMoveAbsolute.Execute		:= FALSE;
				eRunningState							:= E_CapPreScrewer.eReturning2;
			END_IF
			
		END_IF

		
	//Powrót po osi X	
	E_CapPreScrewer.eReturning2:
		bBottleCatcherCatchTemp					:= FALSE;
		bCapsBlowON								:= CartesianZAxisRef.NcToPlc.ActPos > lrAxisZSavedPosition + 10.0;
		
		IF CartesianZAxisRef.NcToPlc.ActPos > stParameters.lrScrewerStartZPosition + 15.0 THEN
			mcCartesianZMoveAbsolute2.Execute		:= TRUE;
			mcCartesianZMoveAbsolute2.Position		:= stParameters.lrTopZPosition;
			mcCartesianZMoveAbsolute2.Acceleration	:= stParameters.lrPickerAcceleration;
			mcCartesianZMoveAbsolute2.Deceleration	:= stParameters.lrPickerAcceleration;
			mcCartesianZMoveAbsolute2.Velocity		:= stParameters.lrPickerSpeed;			
		END_IF
	
		IF (CartesianZAxisRef.NcToPlc.ActPos > stParameters.lrTopZPosition - stParameters.lrBendingDistance) OR
			mcCartesianZMoveAbsolute.Done THEN
			mcCatcherMoveAbsolute.Execute			:= TRUE;		
			mcCatcherMoveAbsolute.Position			:= stParameters.lrCatcherCatchingPosition;
			mcCatcherMoveAbsolute.Acceleration		:= stParameters.lrCatcherAcceleration;
			mcCatcherMoveAbsolute.Deceleration		:= stParameters.lrCatcherAcceleration;
			mcCatcherMoveAbsolute.Velocity			:= stParameters.lrCatcherSpeed;

//SEL(P190_CapFeeder.stMover2Status.bInPlacePosition, GVL_Recipe.lrCapSorterPreScrewerPickXMover1PositionShow, GVL_Recipe.lrCapSorterPreScrewerPickXMover2PositionShow

			
			//Jedź osią poziomą X na pozycję pick
			mcCartesianYMoveAbsolute.Execute		:= TRUE;
			{warning 'Przerobić, dodać parametry obu pozycji wózków do struktury parametrów, FB_CapPreScrewer.Running --> 624'}
			mcCartesianYMoveAbsolute.Position		:= SEL(bMover1InPickPos, GVL_Recipe.lrCapSorterPreScrewerPickXMover1PositionShow, GVL_Recipe.lrCapSorterPreScrewerPickXMover2PositionShow);
			mcCartesianYMoveAbsolute.Acceleration	:= stParameters.lrPickerAcceleration;
			mcCartesianYMoveAbsolute.Deceleration	:= stParameters.lrPickerAcceleration;
			mcCartesianYMoveAbsolute.Velocity		:= stParameters.lrPickerSpeed;
			//Ustaw obracarkę do pozycji początkowej
			
			mcPreScrewerMoveRelative.Distance		:= -1 * DINT_TO_LREAL(LREAL_TO_DINT(PreScrewerAxisRef.NcToPlc.SetPos) MOD 360); 
			mcPreScrewerMoveRelative.Execute		:= mcPreScrewerMoveRelative.Distance<>0 AND NOT mcPreScrewerMoveRelative.Error;
			mcPreScrewerMoveRelative.Acceleration	:= stParameters.lrScrewAcceleration;
			mcPreScrewerMoveRelative.Deceleration	:= stParameters.lrScrewAcceleration;
			mcPreScrewerMoveRelative.Velocity		:= stParameters.lrScrewSpeed;
			
		END_IF
		IF CartesianZAxisRef.NcToPlc.ActPos > stParameters.lrPlaceZPosition + 20 THEN
			bPlaceDone								:= TRUE;
		END_IF
		IF (*bPlaceDone AND*) mcCartesianYMoveAbsolute.Done AND mcCartesianZMoveAbsolute2.Done AND
			 mcCatcherMoveAbsolute.Done THEN
			 IF mcPreScrewerMoveRelative.Distance=0 OR mcPreScrewerMoveRelative.Done THEN
				mcCartesianYMoveAbsolute.Execute		:= FALSE;
 				mcCartesianZMoveAbsolute.Execute		:= FALSE;
				mcCartesianZMoveAbsolute2.Execute		:= FALSE;
				mcCatcherMoveAbsolute.Execute			:= FALSE;
				mcPreScrewerMoveRelative.Execute		:= FALSE;
				eRunningState				:= E_CapPreScrewer.eDone;
			END_IF
		END_IF
		
		//Dodatkowy przedmuch ssawek
		(*IF (CartesianZAxisRef.NcToPlc.ActPos > (stParameters.lrPlaceZPosition + stParameters.lrHeightAdditionalBlow)) THEN
			bAdditionalBlow							S= NOT tonBlowOFF.IN;	
		
			IF NOT bAdditionalBlow THEN
				bCapsBlowON							R= tonBlowOFF.Q;
			END_IF

			bCapsBlowON								S= bAdditionalBlow;
			bCapBlow1 := bCapBlow2 := bCapBlow3 := bCapBlow4 := bAdditionalBlow;
		END_IF*)
			
	E_CapPreScrewer.eDone:
		mcPreScrewerStop.Execute			:= TRUE;
	
		IF mcPreScrewerStop.Done THEN
			mcPreScrewerStop.Execute			:= FALSE;
			bAdditionalBlow						:= FALSE;
			bCycleNotDone						:= FALSE;
			bCapsBlowON							:= FALSE;
			bPlaceDone							:= TRUE;
			bCycleDone							:= TRUE;
			eState								:= E_Station.eDone;
			eRunningState						:= E_CapPreScrewer.eReady;	
		END_IF	

	(*Cykl nie zakończony - przerwany - chyba nie potrzebny*)
	E_CapPreScrewer.eNotDone:
		bCapsBlowON							:= FALSE;
		eState								:= E_Station.eDone;
		eRunningState						:= E_CapPreScrewer.eReady;




END_CASE

tonCapCatcher(PT := T#60MS);
END_ACTION

ACTION RunningWithFlyingSaw:

tonVacuumWatchdog(PT	:= stParameters.tTimeVacuumWatchdog);
bStopAllowed	:= eRunningState = E_CapPreScrewer.eReady OR eRunningState = E_CapPreScrewer.eVerticalDownToCatchPos;

//Otwieranie chwytaków
//bBottleCatcherCatchTemp		R= CartesianZAxisRef.NcToPlc.ActPos < stParameters.lrGripperOpenPosition;
GVL_VIS.bCapSorterPreScrewerBottleCatcherCatch	:= bBottleCatcherCatchTemp AND bCapSorterPreScrewerBottleCatcherEnableShow;
	
tonWaitInPlacePos(PT	:= stParameters.tWaitInPlacePos);
//tonWaitInPlacePos(PT 	:= T#200MS);
eLastRunningState	:= eRunningState;

CASE eRunningState OF

//====================================
	
	(*Oczekiwanie na wykonanie pojedynczego cyklu*)
	E_CapPreScrewer.eReady:

		
		IF NOT bCycleDone AND NOT bCycleNotDone THEN  
                                      	
			IF bRun THEN 
				fbVirtualAxis.fAcceleration				:= stParameters.lrPickerAcceleration;	
				fbVirtualAxis.fDeceleration				:= stParameters.lrPickerAcceleration;	
				fbVirtualAxis.fJerk						:= stParameters.lrPickerJerk;

				iRejectCase					:= 0;
				bRejectDone					:= FALSE;
				bReject						:= FALSE;
				bTubeReject					:= FALSE;
				
				//Przygotuj do cyklu - otwórz chwytaki
				bCapCatcher1				:= FALSE;
				bCapCatcher2				:= FALSE;
				bCapCatcher3				:= FALSE;
				bCapCatcher4				:= FALSE;
	
				//Wyłącz ssawki
				bCapSucker[1]				:= FALSE;
				bCapSucker[2]				:= FALSE;
				bCapSucker[3]				:= FALSE;
				bCapSucker[4]				:= FALSE;
				//Wyłącz odmuchy
				bCapBlower1					:= FALSE;
				bCapBlower2					:= FALSE;
				bCapBlower3					:= FALSE;
				bCapBlower4					:= FALSE;
				bCapsBlowON					:= FALSE;
				//Otwórz chwytaki słomek
				bStrawCatchersOpen			:= TRUE;
				bStrawCatchersClose			:= FALSE;
				//Cofnij chwytaki słomek
				bStrawCatcherActuatorIn		:= TRUE;
				bStrawCatcherActuatorOut	:= FALSE;
				//Podjedź robotem i chwytakiem słomek w górę jak cofnięty chwytak słomek
				IF tonStrawCatcherIn.Q THEN	
										
					mcCartesianZMoveAbsolute.Execute		:= TRUE;		
					mcCartesianZMoveAbsolute.Position		:= stParameters.lrTopZPosition;
					mcCartesianZMoveAbsolute.Acceleration	:= stParameters.lrPickerAcceleration;
					mcCartesianZMoveAbsolute.Deceleration	:= stParameters.lrPickerAcceleration;
					mcCartesianZMoveAbsolute.Velocity		:= stParameters.lrPickerSpeed;
					
					mcCatcherMoveAbsolute.Execute			:= TRUE;		
					mcCatcherMoveAbsolute.Position			:= stParameters.lrCatcherCatchingPosition;
					mcCatcherMoveAbsolute.Acceleration		:= stParameters.lrCatcherAcceleration;
					mcCatcherMoveAbsolute.Deceleration		:= stParameters.lrCatcherAcceleration;
					mcCatcherMoveAbsolute.Velocity			:= stParameters.lrCatcherSpeed;
					
					//Następny krok
					eRunningState						:= E_CapPreScrewer.ePreparingToPick;
					bCycleNotDone						:= TRUE;
					
				END_IF
				//Reset komendy ruchu osi X
				mcCartesianYMoveAbsolute.Execute		:= FALSE;
				
			END_IF
		END_IF
			
	(*Czekam na pozycję Z w górze i ruszam osią poziomą X na pozycję pobierania i czekam na obie pozycje*)
	E_CapPreScrewer.ePreparingToPick:
		IF (CartesianZAxisRef.NcToPlc.ActPos > stParameters.lrTopZPosition - stParameters.lrBendingDistance) OR
			mcCartesianZMoveAbsolute.Done THEN
			//Jedź osią poziomą X na pozycję pick
			mcCartesianYMoveAbsolute.Execute		:= TRUE;
			mcCartesianYMoveAbsolute.Position		:= stParameters.lrPickYPosition;
			mcCartesianYMoveAbsolute.Acceleration	:= stParameters.lrPickerAcceleration;
			mcCartesianYMoveAbsolute.Deceleration	:= stParameters.lrPickerAcceleration;
			mcCartesianYMoveAbsolute.Velocity		:= stParameters.lrPickerSpeed;
			//Nakrętka pobrana z wózka nr.1
			bMover1InPickPos						:= SEL((stParameters.lrPickYPosition-GVL_Recipe.lrCapSorterPreScrewerPickXMover1PositionShow) <= 0.5, FALSE, TRUE);
			
			//Ustaw obracarkę w pozycji
			mcPreScrewerMoveRelative.Distance		:=  -1 * DINT_TO_LREAL((LREAL_TO_DINT(PreScrewerAxisRef.NcToPlc.SetPos)+diPreSCrewerHomePos) MOD 360);
			mcPreScrewerMoveRelative.Execute		:= mcPreScrewerMoveRelative.Distance<>0;
			mcPreScrewerMoveRelative.Acceleration	:= stParameters.lrScrewAcceleration;
			mcPreScrewerMoveRelative.Deceleration	:= stParameters.lrScrewAcceleration;
			mcPreScrewerMoveRelative.Velocity		:= stParameters.lrScrewSpeed;
		END_IF
		//Jak obie pozycje osiągnięte to wysuń chwytak słomek i następny krok
		IF mcCartesianYMoveAbsolute.Done AND mcCartesianZMoveAbsolute.Done AND mcCatcherMoveAbsolute.Done THEN
			IF mcPreScrewerMoveRelative.Done OR mcPreScrewerMoveRelative.Distance =0 THEN
				//Reset komendy ruchu osi
				mcCartesianYMoveAbsolute.Execute		:= FALSE;
				mcCartesianZMoveAbsolute.Execute		:= FALSE;
				mcPreScrewerMoveRelative.Execute		:= FALSE;
				mcCatcherMoveAbsolute.Execute			:= FALSE;
				//Wysuń chwytaki słomek jesli to potrzebuje recepta        
				bStrawCatcherActuatorIn					:= NOT stParameters.bStrawCatcherON;
				bStrawCatcherActuatorOut				:= stParameters.bStrawCatcherON;    
				//Następny krok
				eRunningState							:= E_CapPreScrewer.ePicking;
			END_IF
		END_IF
		
	
